;FOLD SLIN P253 Vel=2 m/s CPDAT253 Tool[4]:Microflown3D Base[2]:straight_sol;%{PE}
;FOLD Parameters ;%{h}
;Params IlfProvider=kukaroboter.basistech.inlineforms.movement.spline; Kuka.IsGlobalPoint=False; Kuka.PointName=P253; Kuka.BlendingEnabled=False; Kuka.MoveDataName=CPDAT253; Kuka.VelocityPath=2.000; Kuka.VelocityFieldEnabled=True; Kuka.ColDetectFieldEnabled=True; Kuka.CurrentCDSetIndex=0; Kuka.MovementParameterFieldEnabled=True; IlfCommand=SLIN
;ENDFOLD
SLIN XP253 WITH $VEL = SVEL_CP(2.0, , LCPDAT253),$TOOL = STOOL2(FP253),$BASE = SBASE(FP253.BASE_NO),$IPO_MODE = SIPO_MODE(FP253.IPO_FRAME),$LOAD = SLOAD(FP253.TOOL_NO),$ACC = SACC_CP(LCPDAT253),$ORI_TYPE = SORI_TYP(LCPDAT253),$APO = SAPO(LCPDAT253),$JERK = SJERK(LCPDAT253),$COLLMON_TOL_PRO[1] = USE_CM_PRO_VALUES(0)
;ENDFOLD

;FOLD SLIN P254 Vel=2 m/s CPDAT254 Tool[4]:Microflown3D Base[2]:straight_sol;%{PE}
;FOLD Parameters ;%{h}
;Params IlfProvider=kukaroboter.basistech.inlineforms.movement.spline; Kuka.IsGlobalPoint=False; Kuka.PointName=P254; Kuka.BlendingEnabled=False; Kuka.MoveDataName=CPDAT254; Kuka.VelocityPath=2.000; Kuka.VelocityFieldEnabled=True; Kuka.ColDetectFieldEnabled=True; Kuka.CurrentCDSetIndex=0; Kuka.MovementParameterFieldEnabled=True; IlfCommand=SLIN
;ENDFOLD
SLIN XP254 WITH $VEL = SVEL_CP(2.0, , LCPDAT254),$TOOL = STOOL2(FP254),$BASE = SBASE(FP254.BASE_NO),$IPO_MODE = SIPO_MODE(FP254.IPO_FRAME),$LOAD = SLOAD(FP254.TOOL_NO),$ACC = SACC_CP(LCPDAT254),$ORI_TYPE = SORI_TYP(LCPDAT254),$APO = SAPO(LCPDAT254),$JERK = SJERK(LCPDAT254),$COLLMON_TOL_PRO[1] = USE_CM_PRO_VALUES(0)
;ENDFOLD

;FOLD SLIN P255 Vel=2 m/s CPDAT255 Tool[4]:Microflown3D Base[2]:straight_sol;%{PE}
;FOLD Parameters ;%{h}
;Params IlfProvider=kukaroboter.basistech.inlineforms.movement.spline; Kuka.IsGlobalPoint=False; Kuka.PointName=P255; Kuka.BlendingEnabled=False; Kuka.MoveDataName=CPDAT255; Kuka.VelocityPath=2.000; Kuka.VelocityFieldEnabled=True; Kuka.ColDetectFieldEnabled=True; Kuka.CurrentCDSetIndex=0; Kuka.MovementParameterFieldEnabled=True; IlfCommand=SLIN
;ENDFOLD
SLIN XP255 WITH $VEL = SVEL_CP(2.0, , LCPDAT255),$TOOL = STOOL2(FP255),$BASE = SBASE(FP255.BASE_NO),$IPO_MODE = SIPO_MODE(FP255.IPO_FRAME),$LOAD = SLOAD(FP255.TOOL_NO),$ACC = SACC_CP(LCPDAT255),$ORI_TYPE = SORI_TYP(LCPDAT255),$APO = SAPO(LCPDAT255),$JERK = SJERK(LCPDAT255),$COLLMON_TOL_PRO[1] = USE_CM_PRO_VALUES(0)
;ENDFOLD

;FOLD SLIN P256 Vel=2 m/s CPDAT256 Tool[4]:Microflown3D Base[2]:straight_sol;%{PE}
;FOLD Parameters ;%{h}
;Params IlfProvider=kukaroboter.basistech.inlineforms.movement.spline; Kuka.IsGlobalPoint=False; Kuka.PointName=P256; Kuka.BlendingEnabled=False; Kuka.MoveDataName=CPDAT256; Kuka.VelocityPath=2.000; Kuka.VelocityFieldEnabled=True; Kuka.ColDetectFieldEnabled=True; Kuka.CurrentCDSetIndex=0; Kuka.MovementParameterFieldEnabled=True; IlfCommand=SLIN
;ENDFOLD
SLIN XP256 WITH $VEL = SVEL_CP(2.0, , LCPDAT256),$TOOL = STOOL2(FP256),$BASE = SBASE(FP256.BASE_NO),$IPO_MODE = SIPO_MODE(FP256.IPO_FRAME),$LOAD = SLOAD(FP256.TOOL_NO),$ACC = SACC_CP(LCPDAT256),$ORI_TYPE = SORI_TYP(LCPDAT256),$APO = SAPO(LCPDAT256),$JERK = SJERK(LCPDAT256),$COLLMON_TOL_PRO[1] = USE_CM_PRO_VALUES(0)
;ENDFOLD

;FOLD SLIN P257 Vel=2 m/s CPDAT257 Tool[4]:Microflown3D Base[2]:straight_sol;%{PE}
;FOLD Parameters ;%{h}
;Params IlfProvider=kukaroboter.basistech.inlineforms.movement.spline; Kuka.IsGlobalPoint=False; Kuka.PointName=P257; Kuka.BlendingEnabled=False; Kuka.MoveDataName=CPDAT257; Kuka.VelocityPath=2.000; Kuka.VelocityFieldEnabled=True; Kuka.ColDetectFieldEnabled=True; Kuka.CurrentCDSetIndex=0; Kuka.MovementParameterFieldEnabled=True; IlfCommand=SLIN
;ENDFOLD
SLIN XP257 WITH $VEL = SVEL_CP(2.0, , LCPDAT257),$TOOL = STOOL2(FP257),$BASE = SBASE(FP257.BASE_NO),$IPO_MODE = SIPO_MODE(FP257.IPO_FRAME),$LOAD = SLOAD(FP257.TOOL_NO),$ACC = SACC_CP(LCPDAT257),$ORI_TYPE = SORI_TYP(LCPDAT257),$APO = SAPO(LCPDAT257),$JERK = SJERK(LCPDAT257),$COLLMON_TOL_PRO[1] = USE_CM_PRO_VALUES(0)
;ENDFOLD

;FOLD SLIN P258 Vel=2 m/s CPDAT258 Tool[4]:Microflown3D Base[2]:straight_sol;%{PE}
;FOLD Parameters ;%{h}
;Params IlfProvider=kukaroboter.basistech.inlineforms.movement.spline; Kuka.IsGlobalPoint=False; Kuka.PointName=P258; Kuka.BlendingEnabled=False; Kuka.MoveDataName=CPDAT258; Kuka.VelocityPath=2.000; Kuka.VelocityFieldEnabled=True; Kuka.ColDetectFieldEnabled=True; Kuka.CurrentCDSetIndex=0; Kuka.MovementParameterFieldEnabled=True; IlfCommand=SLIN
;ENDFOLD
SLIN XP258 WITH $VEL = SVEL_CP(2.0, , LCPDAT258),$TOOL = STOOL2(FP258),$BASE = SBASE(FP258.BASE_NO),$IPO_MODE = SIPO_MODE(FP258.IPO_FRAME),$LOAD = SLOAD(FP258.TOOL_NO),$ACC = SACC_CP(LCPDAT258),$ORI_TYPE = SORI_TYP(LCPDAT258),$APO = SAPO(LCPDAT258),$JERK = SJERK(LCPDAT258),$COLLMON_TOL_PRO[1] = USE_CM_PRO_VALUES(0)
;ENDFOLD

;FOLD SLIN P259 Vel=2 m/s CPDAT259 Tool[4]:Microflown3D Base[2]:straight_sol;%{PE}
;FOLD Parameters ;%{h}
;Params IlfProvider=kukaroboter.basistech.inlineforms.movement.spline; Kuka.IsGlobalPoint=False; Kuka.PointName=P259; Kuka.BlendingEnabled=False; Kuka.MoveDataName=CPDAT259; Kuka.VelocityPath=2.000; Kuka.VelocityFieldEnabled=True; Kuka.ColDetectFieldEnabled=True; Kuka.CurrentCDSetIndex=0; Kuka.MovementParameterFieldEnabled=True; IlfCommand=SLIN
;ENDFOLD
SLIN XP259 WITH $VEL = SVEL_CP(2.0, , LCPDAT259),$TOOL = STOOL2(FP259),$BASE = SBASE(FP259.BASE_NO),$IPO_MODE = SIPO_MODE(FP259.IPO_FRAME),$LOAD = SLOAD(FP259.TOOL_NO),$ACC = SACC_CP(LCPDAT259),$ORI_TYPE = SORI_TYP(LCPDAT259),$APO = SAPO(LCPDAT259),$JERK = SJERK(LCPDAT259),$COLLMON_TOL_PRO[1] = USE_CM_PRO_VALUES(0)
;ENDFOLD

;FOLD SLIN P260 Vel=2 m/s CPDAT260 Tool[4]:Microflown3D Base[2]:straight_sol;%{PE}
;FOLD Parameters ;%{h}
;Params IlfProvider=kukaroboter.basistech.inlineforms.movement.spline; Kuka.IsGlobalPoint=False; Kuka.PointName=P260; Kuka.BlendingEnabled=False; Kuka.MoveDataName=CPDAT260; Kuka.VelocityPath=2.000; Kuka.VelocityFieldEnabled=True; Kuka.ColDetectFieldEnabled=True; Kuka.CurrentCDSetIndex=0; Kuka.MovementParameterFieldEnabled=True; IlfCommand=SLIN
;ENDFOLD
SLIN XP260 WITH $VEL = SVEL_CP(2.0, , LCPDAT260),$TOOL = STOOL2(FP260),$BASE = SBASE(FP260.BASE_NO),$IPO_MODE = SIPO_MODE(FP260.IPO_FRAME),$LOAD = SLOAD(FP260.TOOL_NO),$ACC = SACC_CP(LCPDAT260),$ORI_TYPE = SORI_TYP(LCPDAT260),$APO = SAPO(LCPDAT260),$JERK = SJERK(LCPDAT260),$COLLMON_TOL_PRO[1] = USE_CM_PRO_VALUES(0)
;ENDFOLD

;FOLD SLIN P261 Vel=2 m/s CPDAT261 Tool[4]:Microflown3D Base[2]:straight_sol;%{PE}
;FOLD Parameters ;%{h}
;Params IlfProvider=kukaroboter.basistech.inlineforms.movement.spline; Kuka.IsGlobalPoint=False; Kuka.PointName=P261; Kuka.BlendingEnabled=False; Kuka.MoveDataName=CPDAT261; Kuka.VelocityPath=2.000; Kuka.VelocityFieldEnabled=True; Kuka.ColDetectFieldEnabled=True; Kuka.CurrentCDSetIndex=0; Kuka.MovementParameterFieldEnabled=True; IlfCommand=SLIN
;ENDFOLD
SLIN XP261 WITH $VEL = SVEL_CP(2.0, , LCPDAT261),$TOOL = STOOL2(FP261),$BASE = SBASE(FP261.BASE_NO),$IPO_MODE = SIPO_MODE(FP261.IPO_FRAME),$LOAD = SLOAD(FP261.TOOL_NO),$ACC = SACC_CP(LCPDAT261),$ORI_TYPE = SORI_TYP(LCPDAT261),$APO = SAPO(LCPDAT261),$JERK = SJERK(LCPDAT261),$COLLMON_TOL_PRO[1] = USE_CM_PRO_VALUES(0)
;ENDFOLD

;FOLD SLIN P262 Vel=2 m/s CPDAT262 Tool[4]:Microflown3D Base[2]:straight_sol;%{PE}
;FOLD Parameters ;%{h}
;Params IlfProvider=kukaroboter.basistech.inlineforms.movement.spline; Kuka.IsGlobalPoint=False; Kuka.PointName=P262; Kuka.BlendingEnabled=False; Kuka.MoveDataName=CPDAT262; Kuka.VelocityPath=2.000; Kuka.VelocityFieldEnabled=True; Kuka.ColDetectFieldEnabled=True; Kuka.CurrentCDSetIndex=0; Kuka.MovementParameterFieldEnabled=True; IlfCommand=SLIN
;ENDFOLD
SLIN XP262 WITH $VEL = SVEL_CP(2.0, , LCPDAT262),$TOOL = STOOL2(FP262),$BASE = SBASE(FP262.BASE_NO),$IPO_MODE = SIPO_MODE(FP262.IPO_FRAME),$LOAD = SLOAD(FP262.TOOL_NO),$ACC = SACC_CP(LCPDAT262),$ORI_TYPE = SORI_TYP(LCPDAT262),$APO = SAPO(LCPDAT262),$JERK = SJERK(LCPDAT262),$COLLMON_TOL_PRO[1] = USE_CM_PRO_VALUES(0)
;ENDFOLD

;FOLD SLIN P263 Vel=2 m/s CPDAT263 Tool[4]:Microflown3D Base[2]:straight_sol;%{PE}
;FOLD Parameters ;%{h}
;Params IlfProvider=kukaroboter.basistech.inlineforms.movement.spline; Kuka.IsGlobalPoint=False; Kuka.PointName=P263; Kuka.BlendingEnabled=False; Kuka.MoveDataName=CPDAT263; Kuka.VelocityPath=2.000; Kuka.VelocityFieldEnabled=True; Kuka.ColDetectFieldEnabled=True; Kuka.CurrentCDSetIndex=0; Kuka.MovementParameterFieldEnabled=True; IlfCommand=SLIN
;ENDFOLD
SLIN XP263 WITH $VEL = SVEL_CP(2.0, , LCPDAT263),$TOOL = STOOL2(FP263),$BASE = SBASE(FP263.BASE_NO),$IPO_MODE = SIPO_MODE(FP263.IPO_FRAME),$LOAD = SLOAD(FP263.TOOL_NO),$ACC = SACC_CP(LCPDAT263),$ORI_TYPE = SORI_TYP(LCPDAT263),$APO = SAPO(LCPDAT263),$JERK = SJERK(LCPDAT263),$COLLMON_TOL_PRO[1] = USE_CM_PRO_VALUES(0)
;ENDFOLD

;FOLD SLIN P264 Vel=2 m/s CPDAT264 Tool[4]:Microflown3D Base[2]:straight_sol;%{PE}
;FOLD Parameters ;%{h}
;Params IlfProvider=kukaroboter.basistech.inlineforms.movement.spline; Kuka.IsGlobalPoint=False; Kuka.PointName=P264; Kuka.BlendingEnabled=False; Kuka.MoveDataName=CPDAT264; Kuka.VelocityPath=2.000; Kuka.VelocityFieldEnabled=True; Kuka.ColDetectFieldEnabled=True; Kuka.CurrentCDSetIndex=0; Kuka.MovementParameterFieldEnabled=True; IlfCommand=SLIN
;ENDFOLD
SLIN XP264 WITH $VEL = SVEL_CP(2.0, , LCPDAT264),$TOOL = STOOL2(FP264),$BASE = SBASE(FP264.BASE_NO),$IPO_MODE = SIPO_MODE(FP264.IPO_FRAME),$LOAD = SLOAD(FP264.TOOL_NO),$ACC = SACC_CP(LCPDAT264),$ORI_TYPE = SORI_TYP(LCPDAT264),$APO = SAPO(LCPDAT264),$JERK = SJERK(LCPDAT264),$COLLMON_TOL_PRO[1] = USE_CM_PRO_VALUES(0)
;ENDFOLD

;FOLD SLIN P265 Vel=2 m/s CPDAT265 Tool[4]:Microflown3D Base[2]:straight_sol;%{PE}
;FOLD Parameters ;%{h}
;Params IlfProvider=kukaroboter.basistech.inlineforms.movement.spline; Kuka.IsGlobalPoint=False; Kuka.PointName=P265; Kuka.BlendingEnabled=False; Kuka.MoveDataName=CPDAT265; Kuka.VelocityPath=2.000; Kuka.VelocityFieldEnabled=True; Kuka.ColDetectFieldEnabled=True; Kuka.CurrentCDSetIndex=0; Kuka.MovementParameterFieldEnabled=True; IlfCommand=SLIN
;ENDFOLD
SLIN XP265 WITH $VEL = SVEL_CP(2.0, , LCPDAT265),$TOOL = STOOL2(FP265),$BASE = SBASE(FP265.BASE_NO),$IPO_MODE = SIPO_MODE(FP265.IPO_FRAME),$LOAD = SLOAD(FP265.TOOL_NO),$ACC = SACC_CP(LCPDAT265),$ORI_TYPE = SORI_TYP(LCPDAT265),$APO = SAPO(LCPDAT265),$JERK = SJERK(LCPDAT265),$COLLMON_TOL_PRO[1] = USE_CM_PRO_VALUES(0)
;ENDFOLD

;FOLD SLIN P266 Vel=2 m/s CPDAT266 Tool[4]:Microflown3D Base[2]:straight_sol;%{PE}
;FOLD Parameters ;%{h}
;Params IlfProvider=kukaroboter.basistech.inlineforms.movement.spline; Kuka.IsGlobalPoint=False; Kuka.PointName=P266; Kuka.BlendingEnabled=False; Kuka.MoveDataName=CPDAT266; Kuka.VelocityPath=2.000; Kuka.VelocityFieldEnabled=True; Kuka.ColDetectFieldEnabled=True; Kuka.CurrentCDSetIndex=0; Kuka.MovementParameterFieldEnabled=True; IlfCommand=SLIN
;ENDFOLD
SLIN XP266 WITH $VEL = SVEL_CP(2.0, , LCPDAT266),$TOOL = STOOL2(FP266),$BASE = SBASE(FP266.BASE_NO),$IPO_MODE = SIPO_MODE(FP266.IPO_FRAME),$LOAD = SLOAD(FP266.TOOL_NO),$ACC = SACC_CP(LCPDAT266),$ORI_TYPE = SORI_TYP(LCPDAT266),$APO = SAPO(LCPDAT266),$JERK = SJERK(LCPDAT266),$COLLMON_TOL_PRO[1] = USE_CM_PRO_VALUES(0)
;ENDFOLD

;FOLD SLIN P267 Vel=2 m/s CPDAT267 Tool[4]:Microflown3D Base[2]:straight_sol;%{PE}
;FOLD Parameters ;%{h}
;Params IlfProvider=kukaroboter.basistech.inlineforms.movement.spline; Kuka.IsGlobalPoint=False; Kuka.PointName=P267; Kuka.BlendingEnabled=False; Kuka.MoveDataName=CPDAT267; Kuka.VelocityPath=2.000; Kuka.VelocityFieldEnabled=True; Kuka.ColDetectFieldEnabled=True; Kuka.CurrentCDSetIndex=0; Kuka.MovementParameterFieldEnabled=True; IlfCommand=SLIN
;ENDFOLD
SLIN XP267 WITH $VEL = SVEL_CP(2.0, , LCPDAT267),$TOOL = STOOL2(FP267),$BASE = SBASE(FP267.BASE_NO),$IPO_MODE = SIPO_MODE(FP267.IPO_FRAME),$LOAD = SLOAD(FP267.TOOL_NO),$ACC = SACC_CP(LCPDAT267),$ORI_TYPE = SORI_TYP(LCPDAT267),$APO = SAPO(LCPDAT267),$JERK = SJERK(LCPDAT267),$COLLMON_TOL_PRO[1] = USE_CM_PRO_VALUES(0)
;ENDFOLD

;FOLD SLIN P268 Vel=2 m/s CPDAT268 Tool[4]:Microflown3D Base[2]:straight_sol;%{PE}
;FOLD Parameters ;%{h}
;Params IlfProvider=kukaroboter.basistech.inlineforms.movement.spline; Kuka.IsGlobalPoint=False; Kuka.PointName=P268; Kuka.BlendingEnabled=False; Kuka.MoveDataName=CPDAT268; Kuka.VelocityPath=2.000; Kuka.VelocityFieldEnabled=True; Kuka.ColDetectFieldEnabled=True; Kuka.CurrentCDSetIndex=0; Kuka.MovementParameterFieldEnabled=True; IlfCommand=SLIN
;ENDFOLD
SLIN XP268 WITH $VEL = SVEL_CP(2.0, , LCPDAT268),$TOOL = STOOL2(FP268),$BASE = SBASE(FP268.BASE_NO),$IPO_MODE = SIPO_MODE(FP268.IPO_FRAME),$LOAD = SLOAD(FP268.TOOL_NO),$ACC = SACC_CP(LCPDAT268),$ORI_TYPE = SORI_TYP(LCPDAT268),$APO = SAPO(LCPDAT268),$JERK = SJERK(LCPDAT268),$COLLMON_TOL_PRO[1] = USE_CM_PRO_VALUES(0)
;ENDFOLD

;FOLD SLIN P269 Vel=2 m/s CPDAT269 Tool[4]:Microflown3D Base[2]:straight_sol;%{PE}
;FOLD Parameters ;%{h}
;Params IlfProvider=kukaroboter.basistech.inlineforms.movement.spline; Kuka.IsGlobalPoint=False; Kuka.PointName=P269; Kuka.BlendingEnabled=False; Kuka.MoveDataName=CPDAT269; Kuka.VelocityPath=2.000; Kuka.VelocityFieldEnabled=True; Kuka.ColDetectFieldEnabled=True; Kuka.CurrentCDSetIndex=0; Kuka.MovementParameterFieldEnabled=True; IlfCommand=SLIN
;ENDFOLD
SLIN XP269 WITH $VEL = SVEL_CP(2.0, , LCPDAT269),$TOOL = STOOL2(FP269),$BASE = SBASE(FP269.BASE_NO),$IPO_MODE = SIPO_MODE(FP269.IPO_FRAME),$LOAD = SLOAD(FP269.TOOL_NO),$ACC = SACC_CP(LCPDAT269),$ORI_TYPE = SORI_TYP(LCPDAT269),$APO = SAPO(LCPDAT269),$JERK = SJERK(LCPDAT269),$COLLMON_TOL_PRO[1] = USE_CM_PRO_VALUES(0)
;ENDFOLD

;FOLD SLIN P270 Vel=2 m/s CPDAT270 Tool[4]:Microflown3D Base[2]:straight_sol;%{PE}
;FOLD Parameters ;%{h}
;Params IlfProvider=kukaroboter.basistech.inlineforms.movement.spline; Kuka.IsGlobalPoint=False; Kuka.PointName=P270; Kuka.BlendingEnabled=False; Kuka.MoveDataName=CPDAT270; Kuka.VelocityPath=2.000; Kuka.VelocityFieldEnabled=True; Kuka.ColDetectFieldEnabled=True; Kuka.CurrentCDSetIndex=0; Kuka.MovementParameterFieldEnabled=True; IlfCommand=SLIN
;ENDFOLD
SLIN XP270 WITH $VEL = SVEL_CP(2.0, , LCPDAT270),$TOOL = STOOL2(FP270),$BASE = SBASE(FP270.BASE_NO),$IPO_MODE = SIPO_MODE(FP270.IPO_FRAME),$LOAD = SLOAD(FP270.TOOL_NO),$ACC = SACC_CP(LCPDAT270),$ORI_TYPE = SORI_TYP(LCPDAT270),$APO = SAPO(LCPDAT270),$JERK = SJERK(LCPDAT270),$COLLMON_TOL_PRO[1] = USE_CM_PRO_VALUES(0)
;ENDFOLD

;FOLD SLIN P271 Vel=1 m/s CPDAT271 Tool[4]:Microflown3D Base[2]:straight_sol;%{PE}
;FOLD Parameters ;%{h}
;Params IlfProvider=kukaroboter.basistech.inlineforms.movement.spline; Kuka.IsGlobalPoint=False; Kuka.PointName=P271; Kuka.BlendingEnabled=False; Kuka.MoveDataName=CPDAT271; Kuka.VelocityPath=1.000; Kuka.VelocityFieldEnabled=True; Kuka.ColDetectFieldEnabled=True; Kuka.CurrentCDSetIndex=0; Kuka.MovementParameterFieldEnabled=True; IlfCommand=SLIN
;ENDFOLD
SLIN XP271 WITH $VEL = SVEL_CP(2.0, , LCPDAT271),$TOOL = STOOL2(FP271),$BASE = SBASE(FP271.BASE_NO),$IPO_MODE = SIPO_MODE(FP271.IPO_FRAME),$LOAD = SLOAD(FP271.TOOL_NO),$ACC = SACC_CP(LCPDAT271),$ORI_TYPE = SORI_TYP(LCPDAT271),$APO = SAPO(LCPDAT271),$JERK = SJERK(LCPDAT271),$COLLMON_TOL_PRO[1] = USE_CM_PRO_VALUES(0)
;ENDFOLD

;FOLD SLIN P272 Vel=1 m/s CPDAT272 Tool[4]:Microflown3D Base[2]:straight_sol;%{PE}
;FOLD Parameters ;%{h}
;Params IlfProvider=kukaroboter.basistech.inlineforms.movement.spline; Kuka.IsGlobalPoint=False; Kuka.PointName=P272; Kuka.BlendingEnabled=False; Kuka.MoveDataName=CPDAT272; Kuka.VelocityPath=1.000; Kuka.VelocityFieldEnabled=True; Kuka.ColDetectFieldEnabled=True; Kuka.CurrentCDSetIndex=0; Kuka.MovementParameterFieldEnabled=True; IlfCommand=SLIN
;ENDFOLD
SLIN XP272 WITH $VEL = SVEL_CP(2.0, , LCPDAT272),$TOOL = STOOL2(FP272),$BASE = SBASE(FP272.BASE_NO),$IPO_MODE = SIPO_MODE(FP272.IPO_FRAME),$LOAD = SLOAD(FP272.TOOL_NO),$ACC = SACC_CP(LCPDAT272),$ORI_TYPE = SORI_TYP(LCPDAT272),$APO = SAPO(LCPDAT272),$JERK = SJERK(LCPDAT272),$COLLMON_TOL_PRO[1] = USE_CM_PRO_VALUES(0)
;ENDFOLD

;FOLD SLIN P273 Vel=2 m/s CPDAT273 Tool[4]:Microflown3D Base[2]:straight_sol;%{PE}
;FOLD Parameters ;%{h}
;Params IlfProvider=kukaroboter.basistech.inlineforms.movement.spline; Kuka.IsGlobalPoint=False; Kuka.PointName=P273; Kuka.BlendingEnabled=False; Kuka.MoveDataName=CPDAT273; Kuka.VelocityPath=2.000; Kuka.VelocityFieldEnabled=True; Kuka.ColDetectFieldEnabled=True; Kuka.CurrentCDSetIndex=0; Kuka.MovementParameterFieldEnabled=True; IlfCommand=SLIN
;ENDFOLD
SLIN XP273 WITH $VEL = SVEL_CP(2.0, , LCPDAT273),$TOOL = STOOL2(FP273),$BASE = SBASE(FP273.BASE_NO),$IPO_MODE = SIPO_MODE(FP273.IPO_FRAME),$LOAD = SLOAD(FP273.TOOL_NO),$ACC = SACC_CP(LCPDAT273),$ORI_TYPE = SORI_TYP(LCPDAT273),$APO = SAPO(LCPDAT273),$JERK = SJERK(LCPDAT273),$COLLMON_TOL_PRO[1] = USE_CM_PRO_VALUES(0)
;ENDFOLD

;FOLD SLIN P274 Vel=2 m/s CPDAT274 Tool[4]:Microflown3D Base[2]:straight_sol;%{PE}
;FOLD Parameters ;%{h}
;Params IlfProvider=kukaroboter.basistech.inlineforms.movement.spline; Kuka.IsGlobalPoint=False; Kuka.PointName=P274; Kuka.BlendingEnabled=False; Kuka.MoveDataName=CPDAT274; Kuka.VelocityPath=2.000; Kuka.VelocityFieldEnabled=True; Kuka.ColDetectFieldEnabled=True; Kuka.CurrentCDSetIndex=0; Kuka.MovementParameterFieldEnabled=True; IlfCommand=SLIN
;ENDFOLD
SLIN XP274 WITH $VEL = SVEL_CP(2.0, , LCPDAT274),$TOOL = STOOL2(FP274),$BASE = SBASE(FP274.BASE_NO),$IPO_MODE = SIPO_MODE(FP274.IPO_FRAME),$LOAD = SLOAD(FP274.TOOL_NO),$ACC = SACC_CP(LCPDAT274),$ORI_TYPE = SORI_TYP(LCPDAT274),$APO = SAPO(LCPDAT274),$JERK = SJERK(LCPDAT274),$COLLMON_TOL_PRO[1] = USE_CM_PRO_VALUES(0)
;ENDFOLD

;FOLD SLIN P275 Vel=2 m/s CPDAT275 Tool[4]:Microflown3D Base[2]:straight_sol;%{PE}
;FOLD Parameters ;%{h}
;Params IlfProvider=kukaroboter.basistech.inlineforms.movement.spline; Kuka.IsGlobalPoint=False; Kuka.PointName=P275; Kuka.BlendingEnabled=False; Kuka.MoveDataName=CPDAT275; Kuka.VelocityPath=2.000; Kuka.VelocityFieldEnabled=True; Kuka.ColDetectFieldEnabled=True; Kuka.CurrentCDSetIndex=0; Kuka.MovementParameterFieldEnabled=True; IlfCommand=SLIN
;ENDFOLD
SLIN XP275 WITH $VEL = SVEL_CP(2.0, , LCPDAT275),$TOOL = STOOL2(FP275),$BASE = SBASE(FP275.BASE_NO),$IPO_MODE = SIPO_MODE(FP275.IPO_FRAME),$LOAD = SLOAD(FP275.TOOL_NO),$ACC = SACC_CP(LCPDAT275),$ORI_TYPE = SORI_TYP(LCPDAT275),$APO = SAPO(LCPDAT275),$JERK = SJERK(LCPDAT275),$COLLMON_TOL_PRO[1] = USE_CM_PRO_VALUES(0)
;ENDFOLD

;FOLD SLIN P276 Vel=2 m/s CPDAT276 Tool[4]:Microflown3D Base[2]:straight_sol;%{PE}
;FOLD Parameters ;%{h}
;Params IlfProvider=kukaroboter.basistech.inlineforms.movement.spline; Kuka.IsGlobalPoint=False; Kuka.PointName=P276; Kuka.BlendingEnabled=False; Kuka.MoveDataName=CPDAT276; Kuka.VelocityPath=2.000; Kuka.VelocityFieldEnabled=True; Kuka.ColDetectFieldEnabled=True; Kuka.CurrentCDSetIndex=0; Kuka.MovementParameterFieldEnabled=True; IlfCommand=SLIN
;ENDFOLD
SLIN XP276 WITH $VEL = SVEL_CP(2.0, , LCPDAT276),$TOOL = STOOL2(FP276),$BASE = SBASE(FP276.BASE_NO),$IPO_MODE = SIPO_MODE(FP276.IPO_FRAME),$LOAD = SLOAD(FP276.TOOL_NO),$ACC = SACC_CP(LCPDAT276),$ORI_TYPE = SORI_TYP(LCPDAT276),$APO = SAPO(LCPDAT276),$JERK = SJERK(LCPDAT276),$COLLMON_TOL_PRO[1] = USE_CM_PRO_VALUES(0)
;ENDFOLD

;FOLD SLIN P277 Vel=2 m/s CPDAT277 Tool[4]:Microflown3D Base[2]:straight_sol;%{PE}
;FOLD Parameters ;%{h}
;Params IlfProvider=kukaroboter.basistech.inlineforms.movement.spline; Kuka.IsGlobalPoint=False; Kuka.PointName=P277; Kuka.BlendingEnabled=False; Kuka.MoveDataName=CPDAT277; Kuka.VelocityPath=2.000; Kuka.VelocityFieldEnabled=True; Kuka.ColDetectFieldEnabled=True; Kuka.CurrentCDSetIndex=0; Kuka.MovementParameterFieldEnabled=True; IlfCommand=SLIN
;ENDFOLD
SLIN XP277 WITH $VEL = SVEL_CP(2.0, , LCPDAT277),$TOOL = STOOL2(FP277),$BASE = SBASE(FP277.BASE_NO),$IPO_MODE = SIPO_MODE(FP277.IPO_FRAME),$LOAD = SLOAD(FP277.TOOL_NO),$ACC = SACC_CP(LCPDAT277),$ORI_TYPE = SORI_TYP(LCPDAT277),$APO = SAPO(LCPDAT277),$JERK = SJERK(LCPDAT277),$COLLMON_TOL_PRO[1] = USE_CM_PRO_VALUES(0)
;ENDFOLD

;FOLD SLIN P278 Vel=2 m/s CPDAT278 Tool[4]:Microflown3D Base[2]:straight_sol;%{PE}
;FOLD Parameters ;%{h}
;Params IlfProvider=kukaroboter.basistech.inlineforms.movement.spline; Kuka.IsGlobalPoint=False; Kuka.PointName=P278; Kuka.BlendingEnabled=False; Kuka.MoveDataName=CPDAT278; Kuka.VelocityPath=2.000; Kuka.VelocityFieldEnabled=True; Kuka.ColDetectFieldEnabled=True; Kuka.CurrentCDSetIndex=0; Kuka.MovementParameterFieldEnabled=True; IlfCommand=SLIN
;ENDFOLD
SLIN XP278 WITH $VEL = SVEL_CP(2.0, , LCPDAT278),$TOOL = STOOL2(FP278),$BASE = SBASE(FP278.BASE_NO),$IPO_MODE = SIPO_MODE(FP278.IPO_FRAME),$LOAD = SLOAD(FP278.TOOL_NO),$ACC = SACC_CP(LCPDAT278),$ORI_TYPE = SORI_TYP(LCPDAT278),$APO = SAPO(LCPDAT278),$JERK = SJERK(LCPDAT278),$COLLMON_TOL_PRO[1] = USE_CM_PRO_VALUES(0)
;ENDFOLD

;FOLD SLIN P279 Vel=2 m/s CPDAT279 Tool[4]:Microflown3D Base[2]:straight_sol;%{PE}
;FOLD Parameters ;%{h}
;Params IlfProvider=kukaroboter.basistech.inlineforms.movement.spline; Kuka.IsGlobalPoint=False; Kuka.PointName=P279; Kuka.BlendingEnabled=False; Kuka.MoveDataName=CPDAT279; Kuka.VelocityPath=2.000; Kuka.VelocityFieldEnabled=True; Kuka.ColDetectFieldEnabled=True; Kuka.CurrentCDSetIndex=0; Kuka.MovementParameterFieldEnabled=True; IlfCommand=SLIN
;ENDFOLD
SLIN XP279 WITH $VEL = SVEL_CP(2.0, , LCPDAT279),$TOOL = STOOL2(FP279),$BASE = SBASE(FP279.BASE_NO),$IPO_MODE = SIPO_MODE(FP279.IPO_FRAME),$LOAD = SLOAD(FP279.TOOL_NO),$ACC = SACC_CP(LCPDAT279),$ORI_TYPE = SORI_TYP(LCPDAT279),$APO = SAPO(LCPDAT279),$JERK = SJERK(LCPDAT279),$COLLMON_TOL_PRO[1] = USE_CM_PRO_VALUES(0)
;ENDFOLD

;FOLD SLIN P280 Vel=2 m/s CPDAT280 Tool[4]:Microflown3D Base[2]:straight_sol;%{PE}
;FOLD Parameters ;%{h}
;Params IlfProvider=kukaroboter.basistech.inlineforms.movement.spline; Kuka.IsGlobalPoint=False; Kuka.PointName=P280; Kuka.BlendingEnabled=False; Kuka.MoveDataName=CPDAT280; Kuka.VelocityPath=2.000; Kuka.VelocityFieldEnabled=True; Kuka.ColDetectFieldEnabled=True; Kuka.CurrentCDSetIndex=0; Kuka.MovementParameterFieldEnabled=True; IlfCommand=SLIN
;ENDFOLD
SLIN XP280 WITH $VEL = SVEL_CP(2.0, , LCPDAT280),$TOOL = STOOL2(FP280),$BASE = SBASE(FP280.BASE_NO),$IPO_MODE = SIPO_MODE(FP280.IPO_FRAME),$LOAD = SLOAD(FP280.TOOL_NO),$ACC = SACC_CP(LCPDAT280),$ORI_TYPE = SORI_TYP(LCPDAT280),$APO = SAPO(LCPDAT280),$JERK = SJERK(LCPDAT280),$COLLMON_TOL_PRO[1] = USE_CM_PRO_VALUES(0)
;ENDFOLD

;FOLD SLIN P281 Vel=2 m/s CPDAT281 Tool[4]:Microflown3D Base[2]:straight_sol;%{PE}
;FOLD Parameters ;%{h}
;Params IlfProvider=kukaroboter.basistech.inlineforms.movement.spline; Kuka.IsGlobalPoint=False; Kuka.PointName=P281; Kuka.BlendingEnabled=False; Kuka.MoveDataName=CPDAT281; Kuka.VelocityPath=2.000; Kuka.VelocityFieldEnabled=True; Kuka.ColDetectFieldEnabled=True; Kuka.CurrentCDSetIndex=0; Kuka.MovementParameterFieldEnabled=True; IlfCommand=SLIN
;ENDFOLD
SLIN XP281 WITH $VEL = SVEL_CP(2.0, , LCPDAT281),$TOOL = STOOL2(FP281),$BASE = SBASE(FP281.BASE_NO),$IPO_MODE = SIPO_MODE(FP281.IPO_FRAME),$LOAD = SLOAD(FP281.TOOL_NO),$ACC = SACC_CP(LCPDAT281),$ORI_TYPE = SORI_TYP(LCPDAT281),$APO = SAPO(LCPDAT281),$JERK = SJERK(LCPDAT281),$COLLMON_TOL_PRO[1] = USE_CM_PRO_VALUES(0)
;ENDFOLD

;FOLD SLIN P282 Vel=2 m/s CPDAT282 Tool[4]:Microflown3D Base[2]:straight_sol;%{PE}
;FOLD Parameters ;%{h}
;Params IlfProvider=kukaroboter.basistech.inlineforms.movement.spline; Kuka.IsGlobalPoint=False; Kuka.PointName=P282; Kuka.BlendingEnabled=False; Kuka.MoveDataName=CPDAT282; Kuka.VelocityPath=2.000; Kuka.VelocityFieldEnabled=True; Kuka.ColDetectFieldEnabled=True; Kuka.CurrentCDSetIndex=0; Kuka.MovementParameterFieldEnabled=True; IlfCommand=SLIN
;ENDFOLD
SLIN XP282 WITH $VEL = SVEL_CP(2.0, , LCPDAT282),$TOOL = STOOL2(FP282),$BASE = SBASE(FP282.BASE_NO),$IPO_MODE = SIPO_MODE(FP282.IPO_FRAME),$LOAD = SLOAD(FP282.TOOL_NO),$ACC = SACC_CP(LCPDAT282),$ORI_TYPE = SORI_TYP(LCPDAT282),$APO = SAPO(LCPDAT282),$JERK = SJERK(LCPDAT282),$COLLMON_TOL_PRO[1] = USE_CM_PRO_VALUES(0)
;ENDFOLD

;FOLD SLIN P283 Vel=2 m/s CPDAT283 Tool[4]:Microflown3D Base[2]:straight_sol;%{PE}
;FOLD Parameters ;%{h}
;Params IlfProvider=kukaroboter.basistech.inlineforms.movement.spline; Kuka.IsGlobalPoint=False; Kuka.PointName=P283; Kuka.BlendingEnabled=False; Kuka.MoveDataName=CPDAT283; Kuka.VelocityPath=2.000; Kuka.VelocityFieldEnabled=True; Kuka.ColDetectFieldEnabled=True; Kuka.CurrentCDSetIndex=0; Kuka.MovementParameterFieldEnabled=True; IlfCommand=SLIN
;ENDFOLD
SLIN XP283 WITH $VEL = SVEL_CP(2.0, , LCPDAT283),$TOOL = STOOL2(FP283),$BASE = SBASE(FP283.BASE_NO),$IPO_MODE = SIPO_MODE(FP283.IPO_FRAME),$LOAD = SLOAD(FP283.TOOL_NO),$ACC = SACC_CP(LCPDAT283),$ORI_TYPE = SORI_TYP(LCPDAT283),$APO = SAPO(LCPDAT283),$JERK = SJERK(LCPDAT283),$COLLMON_TOL_PRO[1] = USE_CM_PRO_VALUES(0)
;ENDFOLD

;FOLD SLIN P284 Vel=2 m/s CPDAT284 Tool[4]:Microflown3D Base[2]:straight_sol;%{PE}
;FOLD Parameters ;%{h}
;Params IlfProvider=kukaroboter.basistech.inlineforms.movement.spline; Kuka.IsGlobalPoint=False; Kuka.PointName=P284; Kuka.BlendingEnabled=False; Kuka.MoveDataName=CPDAT284; Kuka.VelocityPath=2.000; Kuka.VelocityFieldEnabled=True; Kuka.ColDetectFieldEnabled=True; Kuka.CurrentCDSetIndex=0; Kuka.MovementParameterFieldEnabled=True; IlfCommand=SLIN
;ENDFOLD
SLIN XP284 WITH $VEL = SVEL_CP(2.0, , LCPDAT284),$TOOL = STOOL2(FP284),$BASE = SBASE(FP284.BASE_NO),$IPO_MODE = SIPO_MODE(FP284.IPO_FRAME),$LOAD = SLOAD(FP284.TOOL_NO),$ACC = SACC_CP(LCPDAT284),$ORI_TYPE = SORI_TYP(LCPDAT284),$APO = SAPO(LCPDAT284),$JERK = SJERK(LCPDAT284),$COLLMON_TOL_PRO[1] = USE_CM_PRO_VALUES(0)
;ENDFOLD

;FOLD SLIN P285 Vel=2 m/s CPDAT285 Tool[4]:Microflown3D Base[2]:straight_sol;%{PE}
;FOLD Parameters ;%{h}
;Params IlfProvider=kukaroboter.basistech.inlineforms.movement.spline; Kuka.IsGlobalPoint=False; Kuka.PointName=P285; Kuka.BlendingEnabled=False; Kuka.MoveDataName=CPDAT285; Kuka.VelocityPath=2.000; Kuka.VelocityFieldEnabled=True; Kuka.ColDetectFieldEnabled=True; Kuka.CurrentCDSetIndex=0; Kuka.MovementParameterFieldEnabled=True; IlfCommand=SLIN
;ENDFOLD
SLIN XP285 WITH $VEL = SVEL_CP(2.0, , LCPDAT285),$TOOL = STOOL2(FP285),$BASE = SBASE(FP285.BASE_NO),$IPO_MODE = SIPO_MODE(FP285.IPO_FRAME),$LOAD = SLOAD(FP285.TOOL_NO),$ACC = SACC_CP(LCPDAT285),$ORI_TYPE = SORI_TYP(LCPDAT285),$APO = SAPO(LCPDAT285),$JERK = SJERK(LCPDAT285),$COLLMON_TOL_PRO[1] = USE_CM_PRO_VALUES(0)
;ENDFOLD

;FOLD SLIN P286 Vel=2 m/s CPDAT286 Tool[4]:Microflown3D Base[2]:straight_sol;%{PE}
;FOLD Parameters ;%{h}
;Params IlfProvider=kukaroboter.basistech.inlineforms.movement.spline; Kuka.IsGlobalPoint=False; Kuka.PointName=P286; Kuka.BlendingEnabled=False; Kuka.MoveDataName=CPDAT286; Kuka.VelocityPath=2.000; Kuka.VelocityFieldEnabled=True; Kuka.ColDetectFieldEnabled=True; Kuka.CurrentCDSetIndex=0; Kuka.MovementParameterFieldEnabled=True; IlfCommand=SLIN
;ENDFOLD
SLIN XP286 WITH $VEL = SVEL_CP(2.0, , LCPDAT286),$TOOL = STOOL2(FP286),$BASE = SBASE(FP286.BASE_NO),$IPO_MODE = SIPO_MODE(FP286.IPO_FRAME),$LOAD = SLOAD(FP286.TOOL_NO),$ACC = SACC_CP(LCPDAT286),$ORI_TYPE = SORI_TYP(LCPDAT286),$APO = SAPO(LCPDAT286),$JERK = SJERK(LCPDAT286),$COLLMON_TOL_PRO[1] = USE_CM_PRO_VALUES(0)
;ENDFOLD

;FOLD SLIN P287 Vel=2 m/s CPDAT287 Tool[4]:Microflown3D Base[2]:straight_sol;%{PE}
;FOLD Parameters ;%{h}
;Params IlfProvider=kukaroboter.basistech.inlineforms.movement.spline; Kuka.IsGlobalPoint=False; Kuka.PointName=P287; Kuka.BlendingEnabled=False; Kuka.MoveDataName=CPDAT287; Kuka.VelocityPath=2.000; Kuka.VelocityFieldEnabled=True; Kuka.ColDetectFieldEnabled=True; Kuka.CurrentCDSetIndex=0; Kuka.MovementParameterFieldEnabled=True; IlfCommand=SLIN
;ENDFOLD
SLIN XP287 WITH $VEL = SVEL_CP(2.0, , LCPDAT287),$TOOL = STOOL2(FP287),$BASE = SBASE(FP287.BASE_NO),$IPO_MODE = SIPO_MODE(FP287.IPO_FRAME),$LOAD = SLOAD(FP287.TOOL_NO),$ACC = SACC_CP(LCPDAT287),$ORI_TYPE = SORI_TYP(LCPDAT287),$APO = SAPO(LCPDAT287),$JERK = SJERK(LCPDAT287),$COLLMON_TOL_PRO[1] = USE_CM_PRO_VALUES(0)
;ENDFOLD

;FOLD SLIN P288 Vel=2 m/s CPDAT288 Tool[4]:Microflown3D Base[2]:straight_sol;%{PE}
;FOLD Parameters ;%{h}
;Params IlfProvider=kukaroboter.basistech.inlineforms.movement.spline; Kuka.IsGlobalPoint=False; Kuka.PointName=P288; Kuka.BlendingEnabled=False; Kuka.MoveDataName=CPDAT288; Kuka.VelocityPath=2.000; Kuka.VelocityFieldEnabled=True; Kuka.ColDetectFieldEnabled=True; Kuka.CurrentCDSetIndex=0; Kuka.MovementParameterFieldEnabled=True; IlfCommand=SLIN
;ENDFOLD
SLIN XP288 WITH $VEL = SVEL_CP(2.0, , LCPDAT288),$TOOL = STOOL2(FP288),$BASE = SBASE(FP288.BASE_NO),$IPO_MODE = SIPO_MODE(FP288.IPO_FRAME),$LOAD = SLOAD(FP288.TOOL_NO),$ACC = SACC_CP(LCPDAT288),$ORI_TYPE = SORI_TYP(LCPDAT288),$APO = SAPO(LCPDAT288),$JERK = SJERK(LCPDAT288),$COLLMON_TOL_PRO[1] = USE_CM_PRO_VALUES(0)
;ENDFOLD

;FOLD SLIN P289 Vel=2 m/s CPDAT289 Tool[4]:Microflown3D Base[2]:straight_sol;%{PE}
;FOLD Parameters ;%{h}
;Params IlfProvider=kukaroboter.basistech.inlineforms.movement.spline; Kuka.IsGlobalPoint=False; Kuka.PointName=P289; Kuka.BlendingEnabled=False; Kuka.MoveDataName=CPDAT289; Kuka.VelocityPath=2.000; Kuka.VelocityFieldEnabled=True; Kuka.ColDetectFieldEnabled=True; Kuka.CurrentCDSetIndex=0; Kuka.MovementParameterFieldEnabled=True; IlfCommand=SLIN
;ENDFOLD
SLIN XP289 WITH $VEL = SVEL_CP(2.0, , LCPDAT289),$TOOL = STOOL2(FP289),$BASE = SBASE(FP289.BASE_NO),$IPO_MODE = SIPO_MODE(FP289.IPO_FRAME),$LOAD = SLOAD(FP289.TOOL_NO),$ACC = SACC_CP(LCPDAT289),$ORI_TYPE = SORI_TYP(LCPDAT289),$APO = SAPO(LCPDAT289),$JERK = SJERK(LCPDAT289),$COLLMON_TOL_PRO[1] = USE_CM_PRO_VALUES(0)
;ENDFOLD

;FOLD SLIN P290 Vel=2 m/s CPDAT290 Tool[4]:Microflown3D Base[2]:straight_sol;%{PE}
;FOLD Parameters ;%{h}
;Params IlfProvider=kukaroboter.basistech.inlineforms.movement.spline; Kuka.IsGlobalPoint=False; Kuka.PointName=P290; Kuka.BlendingEnabled=False; Kuka.MoveDataName=CPDAT290; Kuka.VelocityPath=2.000; Kuka.VelocityFieldEnabled=True; Kuka.ColDetectFieldEnabled=True; Kuka.CurrentCDSetIndex=0; Kuka.MovementParameterFieldEnabled=True; IlfCommand=SLIN
;ENDFOLD
SLIN XP290 WITH $VEL = SVEL_CP(2.0, , LCPDAT290),$TOOL = STOOL2(FP290),$BASE = SBASE(FP290.BASE_NO),$IPO_MODE = SIPO_MODE(FP290.IPO_FRAME),$LOAD = SLOAD(FP290.TOOL_NO),$ACC = SACC_CP(LCPDAT290),$ORI_TYPE = SORI_TYP(LCPDAT290),$APO = SAPO(LCPDAT290),$JERK = SJERK(LCPDAT290),$COLLMON_TOL_PRO[1] = USE_CM_PRO_VALUES(0)
;ENDFOLD

;FOLD SLIN P291 Vel=2 m/s CPDAT291 Tool[4]:Microflown3D Base[2]:straight_sol;%{PE}
;FOLD Parameters ;%{h}
;Params IlfProvider=kukaroboter.basistech.inlineforms.movement.spline; Kuka.IsGlobalPoint=False; Kuka.PointName=P291; Kuka.BlendingEnabled=False; Kuka.MoveDataName=CPDAT291; Kuka.VelocityPath=2.000; Kuka.VelocityFieldEnabled=True; Kuka.ColDetectFieldEnabled=True; Kuka.CurrentCDSetIndex=0; Kuka.MovementParameterFieldEnabled=True; IlfCommand=SLIN
;ENDFOLD
SLIN XP291 WITH $VEL = SVEL_CP(2.0, , LCPDAT291),$TOOL = STOOL2(FP291),$BASE = SBASE(FP291.BASE_NO),$IPO_MODE = SIPO_MODE(FP291.IPO_FRAME),$LOAD = SLOAD(FP291.TOOL_NO),$ACC = SACC_CP(LCPDAT291),$ORI_TYPE = SORI_TYP(LCPDAT291),$APO = SAPO(LCPDAT291),$JERK = SJERK(LCPDAT291),$COLLMON_TOL_PRO[1] = USE_CM_PRO_VALUES(0)
;ENDFOLD

;FOLD SLIN P292 Vel=2 m/s CPDAT292 Tool[4]:Microflown3D Base[2]:straight_sol;%{PE}
;FOLD Parameters ;%{h}
;Params IlfProvider=kukaroboter.basistech.inlineforms.movement.spline; Kuka.IsGlobalPoint=False; Kuka.PointName=P292; Kuka.BlendingEnabled=False; Kuka.MoveDataName=CPDAT292; Kuka.VelocityPath=2.000; Kuka.VelocityFieldEnabled=True; Kuka.ColDetectFieldEnabled=True; Kuka.CurrentCDSetIndex=0; Kuka.MovementParameterFieldEnabled=True; IlfCommand=SLIN
;ENDFOLD
SLIN XP292 WITH $VEL = SVEL_CP(2.0, , LCPDAT292),$TOOL = STOOL2(FP292),$BASE = SBASE(FP292.BASE_NO),$IPO_MODE = SIPO_MODE(FP292.IPO_FRAME),$LOAD = SLOAD(FP292.TOOL_NO),$ACC = SACC_CP(LCPDAT292),$ORI_TYPE = SORI_TYP(LCPDAT292),$APO = SAPO(LCPDAT292),$JERK = SJERK(LCPDAT292),$COLLMON_TOL_PRO[1] = USE_CM_PRO_VALUES(0)
;ENDFOLD

;FOLD SLIN P293 Vel=2 m/s CPDAT293 Tool[4]:Microflown3D Base[2]:straight_sol;%{PE}
;FOLD Parameters ;%{h}
;Params IlfProvider=kukaroboter.basistech.inlineforms.movement.spline; Kuka.IsGlobalPoint=False; Kuka.PointName=P293; Kuka.BlendingEnabled=False; Kuka.MoveDataName=CPDAT293; Kuka.VelocityPath=2.000; Kuka.VelocityFieldEnabled=True; Kuka.ColDetectFieldEnabled=True; Kuka.CurrentCDSetIndex=0; Kuka.MovementParameterFieldEnabled=True; IlfCommand=SLIN
;ENDFOLD
SLIN XP293 WITH $VEL = SVEL_CP(2.0, , LCPDAT293),$TOOL = STOOL2(FP293),$BASE = SBASE(FP293.BASE_NO),$IPO_MODE = SIPO_MODE(FP293.IPO_FRAME),$LOAD = SLOAD(FP293.TOOL_NO),$ACC = SACC_CP(LCPDAT293),$ORI_TYPE = SORI_TYP(LCPDAT293),$APO = SAPO(LCPDAT293),$JERK = SJERK(LCPDAT293),$COLLMON_TOL_PRO[1] = USE_CM_PRO_VALUES(0)
;ENDFOLD

;FOLD SLIN P294 Vel=2 m/s CPDAT294 Tool[4]:Microflown3D Base[2]:straight_sol;%{PE}
;FOLD Parameters ;%{h}
;Params IlfProvider=kukaroboter.basistech.inlineforms.movement.spline; Kuka.IsGlobalPoint=False; Kuka.PointName=P294; Kuka.BlendingEnabled=False; Kuka.MoveDataName=CPDAT294; Kuka.VelocityPath=2.000; Kuka.VelocityFieldEnabled=True; Kuka.ColDetectFieldEnabled=True; Kuka.CurrentCDSetIndex=0; Kuka.MovementParameterFieldEnabled=True; IlfCommand=SLIN
;ENDFOLD
SLIN XP294 WITH $VEL = SVEL_CP(2.0, , LCPDAT294),$TOOL = STOOL2(FP294),$BASE = SBASE(FP294.BASE_NO),$IPO_MODE = SIPO_MODE(FP294.IPO_FRAME),$LOAD = SLOAD(FP294.TOOL_NO),$ACC = SACC_CP(LCPDAT294),$ORI_TYPE = SORI_TYP(LCPDAT294),$APO = SAPO(LCPDAT294),$JERK = SJERK(LCPDAT294),$COLLMON_TOL_PRO[1] = USE_CM_PRO_VALUES(0)
;ENDFOLD

;FOLD SLIN P295 Vel=2 m/s CPDAT295 Tool[4]:Microflown3D Base[2]:straight_sol;%{PE}
;FOLD Parameters ;%{h}
;Params IlfProvider=kukaroboter.basistech.inlineforms.movement.spline; Kuka.IsGlobalPoint=False; Kuka.PointName=P295; Kuka.BlendingEnabled=False; Kuka.MoveDataName=CPDAT295; Kuka.VelocityPath=2.000; Kuka.VelocityFieldEnabled=True; Kuka.ColDetectFieldEnabled=True; Kuka.CurrentCDSetIndex=0; Kuka.MovementParameterFieldEnabled=True; IlfCommand=SLIN
;ENDFOLD
SLIN XP295 WITH $VEL = SVEL_CP(2.0, , LCPDAT295),$TOOL = STOOL2(FP295),$BASE = SBASE(FP295.BASE_NO),$IPO_MODE = SIPO_MODE(FP295.IPO_FRAME),$LOAD = SLOAD(FP295.TOOL_NO),$ACC = SACC_CP(LCPDAT295),$ORI_TYPE = SORI_TYP(LCPDAT295),$APO = SAPO(LCPDAT295),$JERK = SJERK(LCPDAT295),$COLLMON_TOL_PRO[1] = USE_CM_PRO_VALUES(0)
;ENDFOLD

;FOLD SLIN P296 Vel=2 m/s CPDAT296 Tool[4]:Microflown3D Base[2]:straight_sol;%{PE}
;FOLD Parameters ;%{h}
;Params IlfProvider=kukaroboter.basistech.inlineforms.movement.spline; Kuka.IsGlobalPoint=False; Kuka.PointName=P296; Kuka.BlendingEnabled=False; Kuka.MoveDataName=CPDAT296; Kuka.VelocityPath=2.000; Kuka.VelocityFieldEnabled=True; Kuka.ColDetectFieldEnabled=True; Kuka.CurrentCDSetIndex=0; Kuka.MovementParameterFieldEnabled=True; IlfCommand=SLIN
;ENDFOLD
SLIN XP296 WITH $VEL = SVEL_CP(2.0, , LCPDAT296),$TOOL = STOOL2(FP296),$BASE = SBASE(FP296.BASE_NO),$IPO_MODE = SIPO_MODE(FP296.IPO_FRAME),$LOAD = SLOAD(FP296.TOOL_NO),$ACC = SACC_CP(LCPDAT296),$ORI_TYPE = SORI_TYP(LCPDAT296),$APO = SAPO(LCPDAT296),$JERK = SJERK(LCPDAT296),$COLLMON_TOL_PRO[1] = USE_CM_PRO_VALUES(0)
;ENDFOLD

;FOLD SLIN P297 Vel=2 m/s CPDAT297 Tool[4]:Microflown3D Base[2]:straight_sol;%{PE}
;FOLD Parameters ;%{h}
;Params IlfProvider=kukaroboter.basistech.inlineforms.movement.spline; Kuka.IsGlobalPoint=False; Kuka.PointName=P297; Kuka.BlendingEnabled=False; Kuka.MoveDataName=CPDAT297; Kuka.VelocityPath=2.000; Kuka.VelocityFieldEnabled=True; Kuka.ColDetectFieldEnabled=True; Kuka.CurrentCDSetIndex=0; Kuka.MovementParameterFieldEnabled=True; IlfCommand=SLIN
;ENDFOLD
SLIN XP297 WITH $VEL = SVEL_CP(2.0, , LCPDAT297),$TOOL = STOOL2(FP297),$BASE = SBASE(FP297.BASE_NO),$IPO_MODE = SIPO_MODE(FP297.IPO_FRAME),$LOAD = SLOAD(FP297.TOOL_NO),$ACC = SACC_CP(LCPDAT297),$ORI_TYPE = SORI_TYP(LCPDAT297),$APO = SAPO(LCPDAT297),$JERK = SJERK(LCPDAT297),$COLLMON_TOL_PRO[1] = USE_CM_PRO_VALUES(0)
;ENDFOLD

;FOLD SLIN P298 Vel=2 m/s CPDAT298 Tool[4]:Microflown3D Base[2]:straight_sol;%{PE}
;FOLD Parameters ;%{h}
;Params IlfProvider=kukaroboter.basistech.inlineforms.movement.spline; Kuka.IsGlobalPoint=False; Kuka.PointName=P298; Kuka.BlendingEnabled=False; Kuka.MoveDataName=CPDAT298; Kuka.VelocityPath=2.000; Kuka.VelocityFieldEnabled=True; Kuka.ColDetectFieldEnabled=True; Kuka.CurrentCDSetIndex=0; Kuka.MovementParameterFieldEnabled=True; IlfCommand=SLIN
;ENDFOLD
SLIN XP298 WITH $VEL = SVEL_CP(2.0, , LCPDAT298),$TOOL = STOOL2(FP298),$BASE = SBASE(FP298.BASE_NO),$IPO_MODE = SIPO_MODE(FP298.IPO_FRAME),$LOAD = SLOAD(FP298.TOOL_NO),$ACC = SACC_CP(LCPDAT298),$ORI_TYPE = SORI_TYP(LCPDAT298),$APO = SAPO(LCPDAT298),$JERK = SJERK(LCPDAT298),$COLLMON_TOL_PRO[1] = USE_CM_PRO_VALUES(0)
;ENDFOLD

;FOLD SLIN P299 Vel=2 m/s CPDAT299 Tool[4]:Microflown3D Base[2]:straight_sol;%{PE}
;FOLD Parameters ;%{h}
;Params IlfProvider=kukaroboter.basistech.inlineforms.movement.spline; Kuka.IsGlobalPoint=False; Kuka.PointName=P299; Kuka.BlendingEnabled=False; Kuka.MoveDataName=CPDAT299; Kuka.VelocityPath=2.000; Kuka.VelocityFieldEnabled=True; Kuka.ColDetectFieldEnabled=True; Kuka.CurrentCDSetIndex=0; Kuka.MovementParameterFieldEnabled=True; IlfCommand=SLIN
;ENDFOLD
SLIN XP299 WITH $VEL = SVEL_CP(2.0, , LCPDAT299),$TOOL = STOOL2(FP299),$BASE = SBASE(FP299.BASE_NO),$IPO_MODE = SIPO_MODE(FP299.IPO_FRAME),$LOAD = SLOAD(FP299.TOOL_NO),$ACC = SACC_CP(LCPDAT299),$ORI_TYPE = SORI_TYP(LCPDAT299),$APO = SAPO(LCPDAT299),$JERK = SJERK(LCPDAT299),$COLLMON_TOL_PRO[1] = USE_CM_PRO_VALUES(0)
;ENDFOLD

;FOLD SLIN P300 Vel=2 m/s CPDAT300 Tool[4]:Microflown3D Base[2]:straight_sol;%{PE}
;FOLD Parameters ;%{h}
;Params IlfProvider=kukaroboter.basistech.inlineforms.movement.spline; Kuka.IsGlobalPoint=False; Kuka.PointName=P300; Kuka.BlendingEnabled=False; Kuka.MoveDataName=CPDAT300; Kuka.VelocityPath=2.000; Kuka.VelocityFieldEnabled=True; Kuka.ColDetectFieldEnabled=True; Kuka.CurrentCDSetIndex=0; Kuka.MovementParameterFieldEnabled=True; IlfCommand=SLIN
;ENDFOLD
SLIN XP300 WITH $VEL = SVEL_CP(2.0, , LCPDAT300),$TOOL = STOOL2(FP300),$BASE = SBASE(FP300.BASE_NO),$IPO_MODE = SIPO_MODE(FP300.IPO_FRAME),$LOAD = SLOAD(FP300.TOOL_NO),$ACC = SACC_CP(LCPDAT300),$ORI_TYPE = SORI_TYP(LCPDAT300),$APO = SAPO(LCPDAT300),$JERK = SJERK(LCPDAT300),$COLLMON_TOL_PRO[1] = USE_CM_PRO_VALUES(0)
;ENDFOLD

;FOLD SLIN P301 Vel=2 m/s CPDAT301 Tool[4]:Microflown3D Base[2]:straight_sol;%{PE}
;FOLD Parameters ;%{h}
;Params IlfProvider=kukaroboter.basistech.inlineforms.movement.spline; Kuka.IsGlobalPoint=False; Kuka.PointName=P301; Kuka.BlendingEnabled=False; Kuka.MoveDataName=CPDAT301; Kuka.VelocityPath=2.000; Kuka.VelocityFieldEnabled=True; Kuka.ColDetectFieldEnabled=True; Kuka.CurrentCDSetIndex=0; Kuka.MovementParameterFieldEnabled=True; IlfCommand=SLIN
;ENDFOLD
SLIN XP301 WITH $VEL = SVEL_CP(2.0, , LCPDAT301),$TOOL = STOOL2(FP301),$BASE = SBASE(FP301.BASE_NO),$IPO_MODE = SIPO_MODE(FP301.IPO_FRAME),$LOAD = SLOAD(FP301.TOOL_NO),$ACC = SACC_CP(LCPDAT301),$ORI_TYPE = SORI_TYP(LCPDAT301),$APO = SAPO(LCPDAT301),$JERK = SJERK(LCPDAT301),$COLLMON_TOL_PRO[1] = USE_CM_PRO_VALUES(0)
;ENDFOLD

;FOLD SLIN P302 Vel=2 m/s CPDAT302 Tool[4]:Microflown3D Base[2]:straight_sol;%{PE}
;FOLD Parameters ;%{h}
;Params IlfProvider=kukaroboter.basistech.inlineforms.movement.spline; Kuka.IsGlobalPoint=False; Kuka.PointName=P302; Kuka.BlendingEnabled=False; Kuka.MoveDataName=CPDAT302; Kuka.VelocityPath=2.000; Kuka.VelocityFieldEnabled=True; Kuka.ColDetectFieldEnabled=True; Kuka.CurrentCDSetIndex=0; Kuka.MovementParameterFieldEnabled=True; IlfCommand=SLIN
;ENDFOLD
SLIN XP302 WITH $VEL = SVEL_CP(2.0, , LCPDAT302),$TOOL = STOOL2(FP302),$BASE = SBASE(FP302.BASE_NO),$IPO_MODE = SIPO_MODE(FP302.IPO_FRAME),$LOAD = SLOAD(FP302.TOOL_NO),$ACC = SACC_CP(LCPDAT302),$ORI_TYPE = SORI_TYP(LCPDAT302),$APO = SAPO(LCPDAT302),$JERK = SJERK(LCPDAT302),$COLLMON_TOL_PRO[1] = USE_CM_PRO_VALUES(0)
;ENDFOLD

;FOLD SLIN P303 Vel=2 m/s CPDAT303 Tool[4]:Microflown3D Base[2]:straight_sol;%{PE}
;FOLD Parameters ;%{h}
;Params IlfProvider=kukaroboter.basistech.inlineforms.movement.spline; Kuka.IsGlobalPoint=False; Kuka.PointName=P303; Kuka.BlendingEnabled=False; Kuka.MoveDataName=CPDAT303; Kuka.VelocityPath=2.000; Kuka.VelocityFieldEnabled=True; Kuka.ColDetectFieldEnabled=True; Kuka.CurrentCDSetIndex=0; Kuka.MovementParameterFieldEnabled=True; IlfCommand=SLIN
;ENDFOLD
SLIN XP303 WITH $VEL = SVEL_CP(2.0, , LCPDAT303),$TOOL = STOOL2(FP303),$BASE = SBASE(FP303.BASE_NO),$IPO_MODE = SIPO_MODE(FP303.IPO_FRAME),$LOAD = SLOAD(FP303.TOOL_NO),$ACC = SACC_CP(LCPDAT303),$ORI_TYPE = SORI_TYP(LCPDAT303),$APO = SAPO(LCPDAT303),$JERK = SJERK(LCPDAT303),$COLLMON_TOL_PRO[1] = USE_CM_PRO_VALUES(0)
;ENDFOLD

;FOLD SLIN P304 Vel=2 m/s CPDAT304 Tool[4]:Microflown3D Base[2]:straight_sol;%{PE}
;FOLD Parameters ;%{h}
;Params IlfProvider=kukaroboter.basistech.inlineforms.movement.spline; Kuka.IsGlobalPoint=False; Kuka.PointName=P304; Kuka.BlendingEnabled=False; Kuka.MoveDataName=CPDAT304; Kuka.VelocityPath=2.000; Kuka.VelocityFieldEnabled=True; Kuka.ColDetectFieldEnabled=True; Kuka.CurrentCDSetIndex=0; Kuka.MovementParameterFieldEnabled=True; IlfCommand=SLIN
;ENDFOLD
SLIN XP304 WITH $VEL = SVEL_CP(2.0, , LCPDAT304),$TOOL = STOOL2(FP304),$BASE = SBASE(FP304.BASE_NO),$IPO_MODE = SIPO_MODE(FP304.IPO_FRAME),$LOAD = SLOAD(FP304.TOOL_NO),$ACC = SACC_CP(LCPDAT304),$ORI_TYPE = SORI_TYP(LCPDAT304),$APO = SAPO(LCPDAT304),$JERK = SJERK(LCPDAT304),$COLLMON_TOL_PRO[1] = USE_CM_PRO_VALUES(0)
;ENDFOLD

;FOLD SLIN P305 Vel=2 m/s CPDAT305 Tool[4]:Microflown3D Base[2]:straight_sol;%{PE}
;FOLD Parameters ;%{h}
;Params IlfProvider=kukaroboter.basistech.inlineforms.movement.spline; Kuka.IsGlobalPoint=False; Kuka.PointName=P305; Kuka.BlendingEnabled=False; Kuka.MoveDataName=CPDAT305; Kuka.VelocityPath=2.000; Kuka.VelocityFieldEnabled=True; Kuka.ColDetectFieldEnabled=True; Kuka.CurrentCDSetIndex=0; Kuka.MovementParameterFieldEnabled=True; IlfCommand=SLIN
;ENDFOLD
SLIN XP305 WITH $VEL = SVEL_CP(2.0, , LCPDAT305),$TOOL = STOOL2(FP305),$BASE = SBASE(FP305.BASE_NO),$IPO_MODE = SIPO_MODE(FP305.IPO_FRAME),$LOAD = SLOAD(FP305.TOOL_NO),$ACC = SACC_CP(LCPDAT305),$ORI_TYPE = SORI_TYP(LCPDAT305),$APO = SAPO(LCPDAT305),$JERK = SJERK(LCPDAT305),$COLLMON_TOL_PRO[1] = USE_CM_PRO_VALUES(0)
;ENDFOLD

;FOLD SLIN P306 Vel=2 m/s CPDAT306 Tool[4]:Microflown3D Base[2]:straight_sol;%{PE}
;FOLD Parameters ;%{h}
;Params IlfProvider=kukaroboter.basistech.inlineforms.movement.spline; Kuka.IsGlobalPoint=False; Kuka.PointName=P306; Kuka.BlendingEnabled=False; Kuka.MoveDataName=CPDAT306; Kuka.VelocityPath=2.000; Kuka.VelocityFieldEnabled=True; Kuka.ColDetectFieldEnabled=True; Kuka.CurrentCDSetIndex=0; Kuka.MovementParameterFieldEnabled=True; IlfCommand=SLIN
;ENDFOLD
SLIN XP306 WITH $VEL = SVEL_CP(2.0, , LCPDAT306),$TOOL = STOOL2(FP306),$BASE = SBASE(FP306.BASE_NO),$IPO_MODE = SIPO_MODE(FP306.IPO_FRAME),$LOAD = SLOAD(FP306.TOOL_NO),$ACC = SACC_CP(LCPDAT306),$ORI_TYPE = SORI_TYP(LCPDAT306),$APO = SAPO(LCPDAT306),$JERK = SJERK(LCPDAT306),$COLLMON_TOL_PRO[1] = USE_CM_PRO_VALUES(0)
;ENDFOLD

;FOLD SLIN P307 Vel=2 m/s CPDAT307 Tool[4]:Microflown3D Base[2]:straight_sol;%{PE}
;FOLD Parameters ;%{h}
;Params IlfProvider=kukaroboter.basistech.inlineforms.movement.spline; Kuka.IsGlobalPoint=False; Kuka.PointName=P307; Kuka.BlendingEnabled=False; Kuka.MoveDataName=CPDAT307; Kuka.VelocityPath=2.000; Kuka.VelocityFieldEnabled=True; Kuka.ColDetectFieldEnabled=True; Kuka.CurrentCDSetIndex=0; Kuka.MovementParameterFieldEnabled=True; IlfCommand=SLIN
;ENDFOLD
SLIN XP307 WITH $VEL = SVEL_CP(2.0, , LCPDAT307),$TOOL = STOOL2(FP307),$BASE = SBASE(FP307.BASE_NO),$IPO_MODE = SIPO_MODE(FP307.IPO_FRAME),$LOAD = SLOAD(FP307.TOOL_NO),$ACC = SACC_CP(LCPDAT307),$ORI_TYPE = SORI_TYP(LCPDAT307),$APO = SAPO(LCPDAT307),$JERK = SJERK(LCPDAT307),$COLLMON_TOL_PRO[1] = USE_CM_PRO_VALUES(0)
;ENDFOLD

;FOLD SLIN P308 Vel=2 m/s CPDAT308 Tool[4]:Microflown3D Base[2]:straight_sol;%{PE}
;FOLD Parameters ;%{h}
;Params IlfProvider=kukaroboter.basistech.inlineforms.movement.spline; Kuka.IsGlobalPoint=False; Kuka.PointName=P308; Kuka.BlendingEnabled=False; Kuka.MoveDataName=CPDAT308; Kuka.VelocityPath=2.000; Kuka.VelocityFieldEnabled=True; Kuka.ColDetectFieldEnabled=True; Kuka.CurrentCDSetIndex=0; Kuka.MovementParameterFieldEnabled=True; IlfCommand=SLIN
;ENDFOLD
SLIN XP308 WITH $VEL = SVEL_CP(2.0, , LCPDAT308),$TOOL = STOOL2(FP308),$BASE = SBASE(FP308.BASE_NO),$IPO_MODE = SIPO_MODE(FP308.IPO_FRAME),$LOAD = SLOAD(FP308.TOOL_NO),$ACC = SACC_CP(LCPDAT308),$ORI_TYPE = SORI_TYP(LCPDAT308),$APO = SAPO(LCPDAT308),$JERK = SJERK(LCPDAT308),$COLLMON_TOL_PRO[1] = USE_CM_PRO_VALUES(0)
;ENDFOLD

;FOLD SLIN P309 Vel=2 m/s CPDAT309 Tool[4]:Microflown3D Base[2]:straight_sol;%{PE}
;FOLD Parameters ;%{h}
;Params IlfProvider=kukaroboter.basistech.inlineforms.movement.spline; Kuka.IsGlobalPoint=False; Kuka.PointName=P309; Kuka.BlendingEnabled=False; Kuka.MoveDataName=CPDAT309; Kuka.VelocityPath=2.000; Kuka.VelocityFieldEnabled=True; Kuka.ColDetectFieldEnabled=True; Kuka.CurrentCDSetIndex=0; Kuka.MovementParameterFieldEnabled=True; IlfCommand=SLIN
;ENDFOLD
SLIN XP309 WITH $VEL = SVEL_CP(2.0, , LCPDAT309),$TOOL = STOOL2(FP309),$BASE = SBASE(FP309.BASE_NO),$IPO_MODE = SIPO_MODE(FP309.IPO_FRAME),$LOAD = SLOAD(FP309.TOOL_NO),$ACC = SACC_CP(LCPDAT309),$ORI_TYPE = SORI_TYP(LCPDAT309),$APO = SAPO(LCPDAT309),$JERK = SJERK(LCPDAT309),$COLLMON_TOL_PRO[1] = USE_CM_PRO_VALUES(0)
;ENDFOLD

;FOLD SLIN P310 Vel=2 m/s CPDAT310 Tool[4]:Microflown3D Base[2]:straight_sol;%{PE}
;FOLD Parameters ;%{h}
;Params IlfProvider=kukaroboter.basistech.inlineforms.movement.spline; Kuka.IsGlobalPoint=False; Kuka.PointName=P310; Kuka.BlendingEnabled=False; Kuka.MoveDataName=CPDAT310; Kuka.VelocityPath=2.000; Kuka.VelocityFieldEnabled=True; Kuka.ColDetectFieldEnabled=True; Kuka.CurrentCDSetIndex=0; Kuka.MovementParameterFieldEnabled=True; IlfCommand=SLIN
;ENDFOLD
SLIN XP310 WITH $VEL = SVEL_CP(2.0, , LCPDAT310),$TOOL = STOOL2(FP310),$BASE = SBASE(FP310.BASE_NO),$IPO_MODE = SIPO_MODE(FP310.IPO_FRAME),$LOAD = SLOAD(FP310.TOOL_NO),$ACC = SACC_CP(LCPDAT310),$ORI_TYPE = SORI_TYP(LCPDAT310),$APO = SAPO(LCPDAT310),$JERK = SJERK(LCPDAT310),$COLLMON_TOL_PRO[1] = USE_CM_PRO_VALUES(0)
;ENDFOLD

;FOLD SLIN P311 Vel=2 m/s CPDAT311 Tool[4]:Microflown3D Base[2]:straight_sol;%{PE}
;FOLD Parameters ;%{h}
;Params IlfProvider=kukaroboter.basistech.inlineforms.movement.spline; Kuka.IsGlobalPoint=False; Kuka.PointName=P311; Kuka.BlendingEnabled=False; Kuka.MoveDataName=CPDAT311; Kuka.VelocityPath=2.000; Kuka.VelocityFieldEnabled=True; Kuka.ColDetectFieldEnabled=True; Kuka.CurrentCDSetIndex=0; Kuka.MovementParameterFieldEnabled=True; IlfCommand=SLIN
;ENDFOLD
SLIN XP311 WITH $VEL = SVEL_CP(2.0, , LCPDAT311),$TOOL = STOOL2(FP311),$BASE = SBASE(FP311.BASE_NO),$IPO_MODE = SIPO_MODE(FP311.IPO_FRAME),$LOAD = SLOAD(FP311.TOOL_NO),$ACC = SACC_CP(LCPDAT311),$ORI_TYPE = SORI_TYP(LCPDAT311),$APO = SAPO(LCPDAT311),$JERK = SJERK(LCPDAT311),$COLLMON_TOL_PRO[1] = USE_CM_PRO_VALUES(0)
;ENDFOLD

;FOLD SLIN P312 Vel=2 m/s CPDAT312 Tool[4]:Microflown3D Base[2]:straight_sol;%{PE}
;FOLD Parameters ;%{h}
;Params IlfProvider=kukaroboter.basistech.inlineforms.movement.spline; Kuka.IsGlobalPoint=False; Kuka.PointName=P312; Kuka.BlendingEnabled=False; Kuka.MoveDataName=CPDAT312; Kuka.VelocityPath=2.000; Kuka.VelocityFieldEnabled=True; Kuka.ColDetectFieldEnabled=True; Kuka.CurrentCDSetIndex=0; Kuka.MovementParameterFieldEnabled=True; IlfCommand=SLIN
;ENDFOLD
SLIN XP312 WITH $VEL = SVEL_CP(2.0, , LCPDAT312),$TOOL = STOOL2(FP312),$BASE = SBASE(FP312.BASE_NO),$IPO_MODE = SIPO_MODE(FP312.IPO_FRAME),$LOAD = SLOAD(FP312.TOOL_NO),$ACC = SACC_CP(LCPDAT312),$ORI_TYPE = SORI_TYP(LCPDAT312),$APO = SAPO(LCPDAT312),$JERK = SJERK(LCPDAT312),$COLLMON_TOL_PRO[1] = USE_CM_PRO_VALUES(0)
;ENDFOLD

;FOLD SLIN P313 Vel=2 m/s CPDAT313 Tool[4]:Microflown3D Base[2]:straight_sol;%{PE}
;FOLD Parameters ;%{h}
;Params IlfProvider=kukaroboter.basistech.inlineforms.movement.spline; Kuka.IsGlobalPoint=False; Kuka.PointName=P313; Kuka.BlendingEnabled=False; Kuka.MoveDataName=CPDAT313; Kuka.VelocityPath=2.000; Kuka.VelocityFieldEnabled=True; Kuka.ColDetectFieldEnabled=True; Kuka.CurrentCDSetIndex=0; Kuka.MovementParameterFieldEnabled=True; IlfCommand=SLIN
;ENDFOLD
SLIN XP313 WITH $VEL = SVEL_CP(2.0, , LCPDAT313),$TOOL = STOOL2(FP313),$BASE = SBASE(FP313.BASE_NO),$IPO_MODE = SIPO_MODE(FP313.IPO_FRAME),$LOAD = SLOAD(FP313.TOOL_NO),$ACC = SACC_CP(LCPDAT313),$ORI_TYPE = SORI_TYP(LCPDAT313),$APO = SAPO(LCPDAT313),$JERK = SJERK(LCPDAT313),$COLLMON_TOL_PRO[1] = USE_CM_PRO_VALUES(0)
;ENDFOLD

;FOLD SLIN P314 Vel=2 m/s CPDAT314 Tool[4]:Microflown3D Base[2]:straight_sol;%{PE}
;FOLD Parameters ;%{h}
;Params IlfProvider=kukaroboter.basistech.inlineforms.movement.spline; Kuka.IsGlobalPoint=False; Kuka.PointName=P314; Kuka.BlendingEnabled=False; Kuka.MoveDataName=CPDAT314; Kuka.VelocityPath=2.000; Kuka.VelocityFieldEnabled=True; Kuka.ColDetectFieldEnabled=True; Kuka.CurrentCDSetIndex=0; Kuka.MovementParameterFieldEnabled=True; IlfCommand=SLIN
;ENDFOLD
SLIN XP314 WITH $VEL = SVEL_CP(2.0, , LCPDAT314),$TOOL = STOOL2(FP314),$BASE = SBASE(FP314.BASE_NO),$IPO_MODE = SIPO_MODE(FP314.IPO_FRAME),$LOAD = SLOAD(FP314.TOOL_NO),$ACC = SACC_CP(LCPDAT314),$ORI_TYPE = SORI_TYP(LCPDAT314),$APO = SAPO(LCPDAT314),$JERK = SJERK(LCPDAT314),$COLLMON_TOL_PRO[1] = USE_CM_PRO_VALUES(0)
;ENDFOLD

;FOLD SLIN P315 Vel=2 m/s CPDAT315 Tool[4]:Microflown3D Base[2]:straight_sol;%{PE}
;FOLD Parameters ;%{h}
;Params IlfProvider=kukaroboter.basistech.inlineforms.movement.spline; Kuka.IsGlobalPoint=False; Kuka.PointName=P315; Kuka.BlendingEnabled=False; Kuka.MoveDataName=CPDAT315; Kuka.VelocityPath=2.000; Kuka.VelocityFieldEnabled=True; Kuka.ColDetectFieldEnabled=True; Kuka.CurrentCDSetIndex=0; Kuka.MovementParameterFieldEnabled=True; IlfCommand=SLIN
;ENDFOLD
SLIN XP315 WITH $VEL = SVEL_CP(2.0, , LCPDAT315),$TOOL = STOOL2(FP315),$BASE = SBASE(FP315.BASE_NO),$IPO_MODE = SIPO_MODE(FP315.IPO_FRAME),$LOAD = SLOAD(FP315.TOOL_NO),$ACC = SACC_CP(LCPDAT315),$ORI_TYPE = SORI_TYP(LCPDAT315),$APO = SAPO(LCPDAT315),$JERK = SJERK(LCPDAT315),$COLLMON_TOL_PRO[1] = USE_CM_PRO_VALUES(0)
;ENDFOLD

;FOLD SLIN P316 Vel=2 m/s CPDAT316 Tool[4]:Microflown3D Base[2]:straight_sol;%{PE}
;FOLD Parameters ;%{h}
;Params IlfProvider=kukaroboter.basistech.inlineforms.movement.spline; Kuka.IsGlobalPoint=False; Kuka.PointName=P316; Kuka.BlendingEnabled=False; Kuka.MoveDataName=CPDAT316; Kuka.VelocityPath=2.000; Kuka.VelocityFieldEnabled=True; Kuka.ColDetectFieldEnabled=True; Kuka.CurrentCDSetIndex=0; Kuka.MovementParameterFieldEnabled=True; IlfCommand=SLIN
;ENDFOLD
SLIN XP316 WITH $VEL = SVEL_CP(2.0, , LCPDAT316),$TOOL = STOOL2(FP316),$BASE = SBASE(FP316.BASE_NO),$IPO_MODE = SIPO_MODE(FP316.IPO_FRAME),$LOAD = SLOAD(FP316.TOOL_NO),$ACC = SACC_CP(LCPDAT316),$ORI_TYPE = SORI_TYP(LCPDAT316),$APO = SAPO(LCPDAT316),$JERK = SJERK(LCPDAT316),$COLLMON_TOL_PRO[1] = USE_CM_PRO_VALUES(0)
;ENDFOLD

;FOLD SLIN P317 Vel=2 m/s CPDAT317 Tool[4]:Microflown3D Base[2]:straight_sol;%{PE}
;FOLD Parameters ;%{h}
;Params IlfProvider=kukaroboter.basistech.inlineforms.movement.spline; Kuka.IsGlobalPoint=False; Kuka.PointName=P317; Kuka.BlendingEnabled=False; Kuka.MoveDataName=CPDAT317; Kuka.VelocityPath=2.000; Kuka.VelocityFieldEnabled=True; Kuka.ColDetectFieldEnabled=True; Kuka.CurrentCDSetIndex=0; Kuka.MovementParameterFieldEnabled=True; IlfCommand=SLIN
;ENDFOLD
SLIN XP317 WITH $VEL = SVEL_CP(2.0, , LCPDAT317),$TOOL = STOOL2(FP317),$BASE = SBASE(FP317.BASE_NO),$IPO_MODE = SIPO_MODE(FP317.IPO_FRAME),$LOAD = SLOAD(FP317.TOOL_NO),$ACC = SACC_CP(LCPDAT317),$ORI_TYPE = SORI_TYP(LCPDAT317),$APO = SAPO(LCPDAT317),$JERK = SJERK(LCPDAT317),$COLLMON_TOL_PRO[1] = USE_CM_PRO_VALUES(0)
;ENDFOLD

;FOLD SLIN P318 Vel=2 m/s CPDAT318 Tool[4]:Microflown3D Base[2]:straight_sol;%{PE}
;FOLD Parameters ;%{h}
;Params IlfProvider=kukaroboter.basistech.inlineforms.movement.spline; Kuka.IsGlobalPoint=False; Kuka.PointName=P318; Kuka.BlendingEnabled=False; Kuka.MoveDataName=CPDAT318; Kuka.VelocityPath=2.000; Kuka.VelocityFieldEnabled=True; Kuka.ColDetectFieldEnabled=True; Kuka.CurrentCDSetIndex=0; Kuka.MovementParameterFieldEnabled=True; IlfCommand=SLIN
;ENDFOLD
SLIN XP318 WITH $VEL = SVEL_CP(2.0, , LCPDAT318),$TOOL = STOOL2(FP318),$BASE = SBASE(FP318.BASE_NO),$IPO_MODE = SIPO_MODE(FP318.IPO_FRAME),$LOAD = SLOAD(FP318.TOOL_NO),$ACC = SACC_CP(LCPDAT318),$ORI_TYPE = SORI_TYP(LCPDAT318),$APO = SAPO(LCPDAT318),$JERK = SJERK(LCPDAT318),$COLLMON_TOL_PRO[1] = USE_CM_PRO_VALUES(0)
;ENDFOLD

;FOLD SLIN P319 Vel=2 m/s CPDAT319 Tool[4]:Microflown3D Base[2]:straight_sol;%{PE}
;FOLD Parameters ;%{h}
;Params IlfProvider=kukaroboter.basistech.inlineforms.movement.spline; Kuka.IsGlobalPoint=False; Kuka.PointName=P319; Kuka.BlendingEnabled=False; Kuka.MoveDataName=CPDAT319; Kuka.VelocityPath=2.000; Kuka.VelocityFieldEnabled=True; Kuka.ColDetectFieldEnabled=True; Kuka.CurrentCDSetIndex=0; Kuka.MovementParameterFieldEnabled=True; IlfCommand=SLIN
;ENDFOLD
SLIN XP319 WITH $VEL = SVEL_CP(2.0, , LCPDAT319),$TOOL = STOOL2(FP319),$BASE = SBASE(FP319.BASE_NO),$IPO_MODE = SIPO_MODE(FP319.IPO_FRAME),$LOAD = SLOAD(FP319.TOOL_NO),$ACC = SACC_CP(LCPDAT319),$ORI_TYPE = SORI_TYP(LCPDAT319),$APO = SAPO(LCPDAT319),$JERK = SJERK(LCPDAT319),$COLLMON_TOL_PRO[1] = USE_CM_PRO_VALUES(0)
;ENDFOLD

;FOLD SLIN P320 Vel=2 m/s CPDAT320 Tool[4]:Microflown3D Base[2]:straight_sol;%{PE}
;FOLD Parameters ;%{h}
;Params IlfProvider=kukaroboter.basistech.inlineforms.movement.spline; Kuka.IsGlobalPoint=False; Kuka.PointName=P320; Kuka.BlendingEnabled=False; Kuka.MoveDataName=CPDAT320; Kuka.VelocityPath=2.000; Kuka.VelocityFieldEnabled=True; Kuka.ColDetectFieldEnabled=True; Kuka.CurrentCDSetIndex=0; Kuka.MovementParameterFieldEnabled=True; IlfCommand=SLIN
;ENDFOLD
SLIN XP320 WITH $VEL = SVEL_CP(2.0, , LCPDAT320),$TOOL = STOOL2(FP320),$BASE = SBASE(FP320.BASE_NO),$IPO_MODE = SIPO_MODE(FP320.IPO_FRAME),$LOAD = SLOAD(FP320.TOOL_NO),$ACC = SACC_CP(LCPDAT320),$ORI_TYPE = SORI_TYP(LCPDAT320),$APO = SAPO(LCPDAT320),$JERK = SJERK(LCPDAT320),$COLLMON_TOL_PRO[1] = USE_CM_PRO_VALUES(0)
;ENDFOLD

;FOLD SLIN P321 Vel=2 m/s CPDAT321 Tool[4]:Microflown3D Base[2]:straight_sol;%{PE}
;FOLD Parameters ;%{h}
;Params IlfProvider=kukaroboter.basistech.inlineforms.movement.spline; Kuka.IsGlobalPoint=False; Kuka.PointName=P321; Kuka.BlendingEnabled=False; Kuka.MoveDataName=CPDAT321; Kuka.VelocityPath=2.000; Kuka.VelocityFieldEnabled=True; Kuka.ColDetectFieldEnabled=True; Kuka.CurrentCDSetIndex=0; Kuka.MovementParameterFieldEnabled=True; IlfCommand=SLIN
;ENDFOLD
SLIN XP321 WITH $VEL = SVEL_CP(2.0, , LCPDAT321),$TOOL = STOOL2(FP321),$BASE = SBASE(FP321.BASE_NO),$IPO_MODE = SIPO_MODE(FP321.IPO_FRAME),$LOAD = SLOAD(FP321.TOOL_NO),$ACC = SACC_CP(LCPDAT321),$ORI_TYPE = SORI_TYP(LCPDAT321),$APO = SAPO(LCPDAT321),$JERK = SJERK(LCPDAT321),$COLLMON_TOL_PRO[1] = USE_CM_PRO_VALUES(0)
;ENDFOLD

;FOLD SLIN P322 Vel=2 m/s CPDAT322 Tool[4]:Microflown3D Base[2]:straight_sol;%{PE}
;FOLD Parameters ;%{h}
;Params IlfProvider=kukaroboter.basistech.inlineforms.movement.spline; Kuka.IsGlobalPoint=False; Kuka.PointName=P322; Kuka.BlendingEnabled=False; Kuka.MoveDataName=CPDAT322; Kuka.VelocityPath=2.000; Kuka.VelocityFieldEnabled=True; Kuka.ColDetectFieldEnabled=True; Kuka.CurrentCDSetIndex=0; Kuka.MovementParameterFieldEnabled=True; IlfCommand=SLIN
;ENDFOLD
SLIN XP322 WITH $VEL = SVEL_CP(2.0, , LCPDAT322),$TOOL = STOOL2(FP322),$BASE = SBASE(FP322.BASE_NO),$IPO_MODE = SIPO_MODE(FP322.IPO_FRAME),$LOAD = SLOAD(FP322.TOOL_NO),$ACC = SACC_CP(LCPDAT322),$ORI_TYPE = SORI_TYP(LCPDAT322),$APO = SAPO(LCPDAT322),$JERK = SJERK(LCPDAT322),$COLLMON_TOL_PRO[1] = USE_CM_PRO_VALUES(0)
;ENDFOLD

;FOLD SLIN P323 Vel=2 m/s CPDAT323 Tool[4]:Microflown3D Base[2]:straight_sol;%{PE}
;FOLD Parameters ;%{h}
;Params IlfProvider=kukaroboter.basistech.inlineforms.movement.spline; Kuka.IsGlobalPoint=False; Kuka.PointName=P323; Kuka.BlendingEnabled=False; Kuka.MoveDataName=CPDAT323; Kuka.VelocityPath=2.000; Kuka.VelocityFieldEnabled=True; Kuka.ColDetectFieldEnabled=True; Kuka.CurrentCDSetIndex=0; Kuka.MovementParameterFieldEnabled=True; IlfCommand=SLIN
;ENDFOLD
SLIN XP323 WITH $VEL = SVEL_CP(2.0, , LCPDAT323),$TOOL = STOOL2(FP323),$BASE = SBASE(FP323.BASE_NO),$IPO_MODE = SIPO_MODE(FP323.IPO_FRAME),$LOAD = SLOAD(FP323.TOOL_NO),$ACC = SACC_CP(LCPDAT323),$ORI_TYPE = SORI_TYP(LCPDAT323),$APO = SAPO(LCPDAT323),$JERK = SJERK(LCPDAT323),$COLLMON_TOL_PRO[1] = USE_CM_PRO_VALUES(0)
;ENDFOLD

;FOLD SLIN P324 Vel=2 m/s CPDAT324 Tool[4]:Microflown3D Base[2]:straight_sol;%{PE}
;FOLD Parameters ;%{h}
;Params IlfProvider=kukaroboter.basistech.inlineforms.movement.spline; Kuka.IsGlobalPoint=False; Kuka.PointName=P324; Kuka.BlendingEnabled=False; Kuka.MoveDataName=CPDAT324; Kuka.VelocityPath=2.000; Kuka.VelocityFieldEnabled=True; Kuka.ColDetectFieldEnabled=True; Kuka.CurrentCDSetIndex=0; Kuka.MovementParameterFieldEnabled=True; IlfCommand=SLIN
;ENDFOLD
SLIN XP324 WITH $VEL = SVEL_CP(2.0, , LCPDAT324),$TOOL = STOOL2(FP324),$BASE = SBASE(FP324.BASE_NO),$IPO_MODE = SIPO_MODE(FP324.IPO_FRAME),$LOAD = SLOAD(FP324.TOOL_NO),$ACC = SACC_CP(LCPDAT324),$ORI_TYPE = SORI_TYP(LCPDAT324),$APO = SAPO(LCPDAT324),$JERK = SJERK(LCPDAT324),$COLLMON_TOL_PRO[1] = USE_CM_PRO_VALUES(0)
;ENDFOLD

;FOLD SLIN P325 Vel=2 m/s CPDAT325 Tool[4]:Microflown3D Base[2]:straight_sol;%{PE}
;FOLD Parameters ;%{h}
;Params IlfProvider=kukaroboter.basistech.inlineforms.movement.spline; Kuka.IsGlobalPoint=False; Kuka.PointName=P325; Kuka.BlendingEnabled=False; Kuka.MoveDataName=CPDAT325; Kuka.VelocityPath=2.000; Kuka.VelocityFieldEnabled=True; Kuka.ColDetectFieldEnabled=True; Kuka.CurrentCDSetIndex=0; Kuka.MovementParameterFieldEnabled=True; IlfCommand=SLIN
;ENDFOLD
SLIN XP325 WITH $VEL = SVEL_CP(2.0, , LCPDAT325),$TOOL = STOOL2(FP325),$BASE = SBASE(FP325.BASE_NO),$IPO_MODE = SIPO_MODE(FP325.IPO_FRAME),$LOAD = SLOAD(FP325.TOOL_NO),$ACC = SACC_CP(LCPDAT325),$ORI_TYPE = SORI_TYP(LCPDAT325),$APO = SAPO(LCPDAT325),$JERK = SJERK(LCPDAT325),$COLLMON_TOL_PRO[1] = USE_CM_PRO_VALUES(0)
;ENDFOLD

;FOLD SLIN P326 Vel=2 m/s CPDAT326 Tool[4]:Microflown3D Base[2]:straight_sol;%{PE}
;FOLD Parameters ;%{h}
;Params IlfProvider=kukaroboter.basistech.inlineforms.movement.spline; Kuka.IsGlobalPoint=False; Kuka.PointName=P326; Kuka.BlendingEnabled=False; Kuka.MoveDataName=CPDAT326; Kuka.VelocityPath=2.000; Kuka.VelocityFieldEnabled=True; Kuka.ColDetectFieldEnabled=True; Kuka.CurrentCDSetIndex=0; Kuka.MovementParameterFieldEnabled=True; IlfCommand=SLIN
;ENDFOLD
SLIN XP326 WITH $VEL = SVEL_CP(2.0, , LCPDAT326),$TOOL = STOOL2(FP326),$BASE = SBASE(FP326.BASE_NO),$IPO_MODE = SIPO_MODE(FP326.IPO_FRAME),$LOAD = SLOAD(FP326.TOOL_NO),$ACC = SACC_CP(LCPDAT326),$ORI_TYPE = SORI_TYP(LCPDAT326),$APO = SAPO(LCPDAT326),$JERK = SJERK(LCPDAT326),$COLLMON_TOL_PRO[1] = USE_CM_PRO_VALUES(0)
;ENDFOLD

;FOLD SLIN P327 Vel=2 m/s CPDAT327 Tool[4]:Microflown3D Base[2]:straight_sol;%{PE}
;FOLD Parameters ;%{h}
;Params IlfProvider=kukaroboter.basistech.inlineforms.movement.spline; Kuka.IsGlobalPoint=False; Kuka.PointName=P327; Kuka.BlendingEnabled=False; Kuka.MoveDataName=CPDAT327; Kuka.VelocityPath=2.000; Kuka.VelocityFieldEnabled=True; Kuka.ColDetectFieldEnabled=True; Kuka.CurrentCDSetIndex=0; Kuka.MovementParameterFieldEnabled=True; IlfCommand=SLIN
;ENDFOLD
SLIN XP327 WITH $VEL = SVEL_CP(2.0, , LCPDAT327),$TOOL = STOOL2(FP327),$BASE = SBASE(FP327.BASE_NO),$IPO_MODE = SIPO_MODE(FP327.IPO_FRAME),$LOAD = SLOAD(FP327.TOOL_NO),$ACC = SACC_CP(LCPDAT327),$ORI_TYPE = SORI_TYP(LCPDAT327),$APO = SAPO(LCPDAT327),$JERK = SJERK(LCPDAT327),$COLLMON_TOL_PRO[1] = USE_CM_PRO_VALUES(0)
;ENDFOLD

;FOLD SLIN P328 Vel=2 m/s CPDAT328 Tool[4]:Microflown3D Base[2]:straight_sol;%{PE}
;FOLD Parameters ;%{h}
;Params IlfProvider=kukaroboter.basistech.inlineforms.movement.spline; Kuka.IsGlobalPoint=False; Kuka.PointName=P328; Kuka.BlendingEnabled=False; Kuka.MoveDataName=CPDAT328; Kuka.VelocityPath=2.000; Kuka.VelocityFieldEnabled=True; Kuka.ColDetectFieldEnabled=True; Kuka.CurrentCDSetIndex=0; Kuka.MovementParameterFieldEnabled=True; IlfCommand=SLIN
;ENDFOLD
SLIN XP328 WITH $VEL = SVEL_CP(2.0, , LCPDAT328),$TOOL = STOOL2(FP328),$BASE = SBASE(FP328.BASE_NO),$IPO_MODE = SIPO_MODE(FP328.IPO_FRAME),$LOAD = SLOAD(FP328.TOOL_NO),$ACC = SACC_CP(LCPDAT328),$ORI_TYPE = SORI_TYP(LCPDAT328),$APO = SAPO(LCPDAT328),$JERK = SJERK(LCPDAT328),$COLLMON_TOL_PRO[1] = USE_CM_PRO_VALUES(0)
;ENDFOLD

;FOLD SLIN P329 Vel=2 m/s CPDAT329 Tool[4]:Microflown3D Base[2]:straight_sol;%{PE}
;FOLD Parameters ;%{h}
;Params IlfProvider=kukaroboter.basistech.inlineforms.movement.spline; Kuka.IsGlobalPoint=False; Kuka.PointName=P329; Kuka.BlendingEnabled=False; Kuka.MoveDataName=CPDAT329; Kuka.VelocityPath=2.000; Kuka.VelocityFieldEnabled=True; Kuka.ColDetectFieldEnabled=True; Kuka.CurrentCDSetIndex=0; Kuka.MovementParameterFieldEnabled=True; IlfCommand=SLIN
;ENDFOLD
SLIN XP329 WITH $VEL = SVEL_CP(2.0, , LCPDAT329),$TOOL = STOOL2(FP329),$BASE = SBASE(FP329.BASE_NO),$IPO_MODE = SIPO_MODE(FP329.IPO_FRAME),$LOAD = SLOAD(FP329.TOOL_NO),$ACC = SACC_CP(LCPDAT329),$ORI_TYPE = SORI_TYP(LCPDAT329),$APO = SAPO(LCPDAT329),$JERK = SJERK(LCPDAT329),$COLLMON_TOL_PRO[1] = USE_CM_PRO_VALUES(0)
;ENDFOLD

;FOLD SLIN P330 Vel=2 m/s CPDAT330 Tool[4]:Microflown3D Base[2]:straight_sol;%{PE}
;FOLD Parameters ;%{h}
;Params IlfProvider=kukaroboter.basistech.inlineforms.movement.spline; Kuka.IsGlobalPoint=False; Kuka.PointName=P330; Kuka.BlendingEnabled=False; Kuka.MoveDataName=CPDAT330; Kuka.VelocityPath=2.000; Kuka.VelocityFieldEnabled=True; Kuka.ColDetectFieldEnabled=True; Kuka.CurrentCDSetIndex=0; Kuka.MovementParameterFieldEnabled=True; IlfCommand=SLIN
;ENDFOLD
SLIN XP330 WITH $VEL = SVEL_CP(2.0, , LCPDAT330),$TOOL = STOOL2(FP330),$BASE = SBASE(FP330.BASE_NO),$IPO_MODE = SIPO_MODE(FP330.IPO_FRAME),$LOAD = SLOAD(FP330.TOOL_NO),$ACC = SACC_CP(LCPDAT330),$ORI_TYPE = SORI_TYP(LCPDAT330),$APO = SAPO(LCPDAT330),$JERK = SJERK(LCPDAT330),$COLLMON_TOL_PRO[1] = USE_CM_PRO_VALUES(0)
;ENDFOLD

;FOLD SLIN P331 Vel=2 m/s CPDAT331 Tool[4]:Microflown3D Base[2]:straight_sol;%{PE}
;FOLD Parameters ;%{h}
;Params IlfProvider=kukaroboter.basistech.inlineforms.movement.spline; Kuka.IsGlobalPoint=False; Kuka.PointName=P331; Kuka.BlendingEnabled=False; Kuka.MoveDataName=CPDAT331; Kuka.VelocityPath=2.000; Kuka.VelocityFieldEnabled=True; Kuka.ColDetectFieldEnabled=True; Kuka.CurrentCDSetIndex=0; Kuka.MovementParameterFieldEnabled=True; IlfCommand=SLIN
;ENDFOLD
SLIN XP331 WITH $VEL = SVEL_CP(2.0, , LCPDAT331),$TOOL = STOOL2(FP331),$BASE = SBASE(FP331.BASE_NO),$IPO_MODE = SIPO_MODE(FP331.IPO_FRAME),$LOAD = SLOAD(FP331.TOOL_NO),$ACC = SACC_CP(LCPDAT331),$ORI_TYPE = SORI_TYP(LCPDAT331),$APO = SAPO(LCPDAT331),$JERK = SJERK(LCPDAT331),$COLLMON_TOL_PRO[1] = USE_CM_PRO_VALUES(0)
;ENDFOLD

;FOLD SLIN P332 Vel=2 m/s CPDAT332 Tool[4]:Microflown3D Base[2]:straight_sol;%{PE}
;FOLD Parameters ;%{h}
;Params IlfProvider=kukaroboter.basistech.inlineforms.movement.spline; Kuka.IsGlobalPoint=False; Kuka.PointName=P332; Kuka.BlendingEnabled=False; Kuka.MoveDataName=CPDAT332; Kuka.VelocityPath=2.000; Kuka.VelocityFieldEnabled=True; Kuka.ColDetectFieldEnabled=True; Kuka.CurrentCDSetIndex=0; Kuka.MovementParameterFieldEnabled=True; IlfCommand=SLIN
;ENDFOLD
SLIN XP332 WITH $VEL = SVEL_CP(2.0, , LCPDAT332),$TOOL = STOOL2(FP332),$BASE = SBASE(FP332.BASE_NO),$IPO_MODE = SIPO_MODE(FP332.IPO_FRAME),$LOAD = SLOAD(FP332.TOOL_NO),$ACC = SACC_CP(LCPDAT332),$ORI_TYPE = SORI_TYP(LCPDAT332),$APO = SAPO(LCPDAT332),$JERK = SJERK(LCPDAT332),$COLLMON_TOL_PRO[1] = USE_CM_PRO_VALUES(0)
;ENDFOLD

;FOLD SLIN P333 Vel=2 m/s CPDAT333 Tool[4]:Microflown3D Base[2]:straight_sol;%{PE}
;FOLD Parameters ;%{h}
;Params IlfProvider=kukaroboter.basistech.inlineforms.movement.spline; Kuka.IsGlobalPoint=False; Kuka.PointName=P333; Kuka.BlendingEnabled=False; Kuka.MoveDataName=CPDAT333; Kuka.VelocityPath=2.000; Kuka.VelocityFieldEnabled=True; Kuka.ColDetectFieldEnabled=True; Kuka.CurrentCDSetIndex=0; Kuka.MovementParameterFieldEnabled=True; IlfCommand=SLIN
;ENDFOLD
SLIN XP333 WITH $VEL = SVEL_CP(2.0, , LCPDAT333),$TOOL = STOOL2(FP333),$BASE = SBASE(FP333.BASE_NO),$IPO_MODE = SIPO_MODE(FP333.IPO_FRAME),$LOAD = SLOAD(FP333.TOOL_NO),$ACC = SACC_CP(LCPDAT333),$ORI_TYPE = SORI_TYP(LCPDAT333),$APO = SAPO(LCPDAT333),$JERK = SJERK(LCPDAT333),$COLLMON_TOL_PRO[1] = USE_CM_PRO_VALUES(0)
;ENDFOLD

;FOLD SLIN P334 Vel=2 m/s CPDAT334 Tool[4]:Microflown3D Base[2]:straight_sol;%{PE}
;FOLD Parameters ;%{h}
;Params IlfProvider=kukaroboter.basistech.inlineforms.movement.spline; Kuka.IsGlobalPoint=False; Kuka.PointName=P334; Kuka.BlendingEnabled=False; Kuka.MoveDataName=CPDAT334; Kuka.VelocityPath=2.000; Kuka.VelocityFieldEnabled=True; Kuka.ColDetectFieldEnabled=True; Kuka.CurrentCDSetIndex=0; Kuka.MovementParameterFieldEnabled=True; IlfCommand=SLIN
;ENDFOLD
SLIN XP334 WITH $VEL = SVEL_CP(2.0, , LCPDAT334),$TOOL = STOOL2(FP334),$BASE = SBASE(FP334.BASE_NO),$IPO_MODE = SIPO_MODE(FP334.IPO_FRAME),$LOAD = SLOAD(FP334.TOOL_NO),$ACC = SACC_CP(LCPDAT334),$ORI_TYPE = SORI_TYP(LCPDAT334),$APO = SAPO(LCPDAT334),$JERK = SJERK(LCPDAT334),$COLLMON_TOL_PRO[1] = USE_CM_PRO_VALUES(0)
;ENDFOLD

;FOLD SLIN P335 Vel=2 m/s CPDAT335 Tool[4]:Microflown3D Base[2]:straight_sol;%{PE}
;FOLD Parameters ;%{h}
;Params IlfProvider=kukaroboter.basistech.inlineforms.movement.spline; Kuka.IsGlobalPoint=False; Kuka.PointName=P335; Kuka.BlendingEnabled=False; Kuka.MoveDataName=CPDAT335; Kuka.VelocityPath=2.000; Kuka.VelocityFieldEnabled=True; Kuka.ColDetectFieldEnabled=True; Kuka.CurrentCDSetIndex=0; Kuka.MovementParameterFieldEnabled=True; IlfCommand=SLIN
;ENDFOLD
SLIN XP335 WITH $VEL = SVEL_CP(2.0, , LCPDAT335),$TOOL = STOOL2(FP335),$BASE = SBASE(FP335.BASE_NO),$IPO_MODE = SIPO_MODE(FP335.IPO_FRAME),$LOAD = SLOAD(FP335.TOOL_NO),$ACC = SACC_CP(LCPDAT335),$ORI_TYPE = SORI_TYP(LCPDAT335),$APO = SAPO(LCPDAT335),$JERK = SJERK(LCPDAT335),$COLLMON_TOL_PRO[1] = USE_CM_PRO_VALUES(0)
;ENDFOLD

;FOLD SLIN P336 Vel=2 m/s CPDAT336 Tool[4]:Microflown3D Base[2]:straight_sol;%{PE}
;FOLD Parameters ;%{h}
;Params IlfProvider=kukaroboter.basistech.inlineforms.movement.spline; Kuka.IsGlobalPoint=False; Kuka.PointName=P336; Kuka.BlendingEnabled=False; Kuka.MoveDataName=CPDAT336; Kuka.VelocityPath=2.000; Kuka.VelocityFieldEnabled=True; Kuka.ColDetectFieldEnabled=True; Kuka.CurrentCDSetIndex=0; Kuka.MovementParameterFieldEnabled=True; IlfCommand=SLIN
;ENDFOLD
SLIN XP336 WITH $VEL = SVEL_CP(2.0, , LCPDAT336),$TOOL = STOOL2(FP336),$BASE = SBASE(FP336.BASE_NO),$IPO_MODE = SIPO_MODE(FP336.IPO_FRAME),$LOAD = SLOAD(FP336.TOOL_NO),$ACC = SACC_CP(LCPDAT336),$ORI_TYPE = SORI_TYP(LCPDAT336),$APO = SAPO(LCPDAT336),$JERK = SJERK(LCPDAT336),$COLLMON_TOL_PRO[1] = USE_CM_PRO_VALUES(0)
;ENDFOLD

;FOLD SLIN P337 Vel=2 m/s CPDAT337 Tool[4]:Microflown3D Base[2]:straight_sol;%{PE}
;FOLD Parameters ;%{h}
;Params IlfProvider=kukaroboter.basistech.inlineforms.movement.spline; Kuka.IsGlobalPoint=False; Kuka.PointName=P337; Kuka.BlendingEnabled=False; Kuka.MoveDataName=CPDAT337; Kuka.VelocityPath=2.000; Kuka.VelocityFieldEnabled=True; Kuka.ColDetectFieldEnabled=True; Kuka.CurrentCDSetIndex=0; Kuka.MovementParameterFieldEnabled=True; IlfCommand=SLIN
;ENDFOLD
SLIN XP337 WITH $VEL = SVEL_CP(2.0, , LCPDAT337),$TOOL = STOOL2(FP337),$BASE = SBASE(FP337.BASE_NO),$IPO_MODE = SIPO_MODE(FP337.IPO_FRAME),$LOAD = SLOAD(FP337.TOOL_NO),$ACC = SACC_CP(LCPDAT337),$ORI_TYPE = SORI_TYP(LCPDAT337),$APO = SAPO(LCPDAT337),$JERK = SJERK(LCPDAT337),$COLLMON_TOL_PRO[1] = USE_CM_PRO_VALUES(0)
;ENDFOLD

;FOLD SLIN P338 Vel=2 m/s CPDAT338 Tool[4]:Microflown3D Base[2]:straight_sol;%{PE}
;FOLD Parameters ;%{h}
;Params IlfProvider=kukaroboter.basistech.inlineforms.movement.spline; Kuka.IsGlobalPoint=False; Kuka.PointName=P338; Kuka.BlendingEnabled=False; Kuka.MoveDataName=CPDAT338; Kuka.VelocityPath=2.000; Kuka.VelocityFieldEnabled=True; Kuka.ColDetectFieldEnabled=True; Kuka.CurrentCDSetIndex=0; Kuka.MovementParameterFieldEnabled=True; IlfCommand=SLIN
;ENDFOLD
SLIN XP338 WITH $VEL = SVEL_CP(2.0, , LCPDAT338),$TOOL = STOOL2(FP338),$BASE = SBASE(FP338.BASE_NO),$IPO_MODE = SIPO_MODE(FP338.IPO_FRAME),$LOAD = SLOAD(FP338.TOOL_NO),$ACC = SACC_CP(LCPDAT338),$ORI_TYPE = SORI_TYP(LCPDAT338),$APO = SAPO(LCPDAT338),$JERK = SJERK(LCPDAT338),$COLLMON_TOL_PRO[1] = USE_CM_PRO_VALUES(0)
;ENDFOLD

;FOLD SLIN P339 Vel=2 m/s CPDAT339 Tool[4]:Microflown3D Base[2]:straight_sol;%{PE}
;FOLD Parameters ;%{h}
;Params IlfProvider=kukaroboter.basistech.inlineforms.movement.spline; Kuka.IsGlobalPoint=False; Kuka.PointName=P339; Kuka.BlendingEnabled=False; Kuka.MoveDataName=CPDAT339; Kuka.VelocityPath=2.000; Kuka.VelocityFieldEnabled=True; Kuka.ColDetectFieldEnabled=True; Kuka.CurrentCDSetIndex=0; Kuka.MovementParameterFieldEnabled=True; IlfCommand=SLIN
;ENDFOLD
SLIN XP339 WITH $VEL = SVEL_CP(2.0, , LCPDAT339),$TOOL = STOOL2(FP339),$BASE = SBASE(FP339.BASE_NO),$IPO_MODE = SIPO_MODE(FP339.IPO_FRAME),$LOAD = SLOAD(FP339.TOOL_NO),$ACC = SACC_CP(LCPDAT339),$ORI_TYPE = SORI_TYP(LCPDAT339),$APO = SAPO(LCPDAT339),$JERK = SJERK(LCPDAT339),$COLLMON_TOL_PRO[1] = USE_CM_PRO_VALUES(0)
;ENDFOLD

;FOLD SLIN P340 Vel=2 m/s CPDAT340 Tool[4]:Microflown3D Base[2]:straight_sol;%{PE}
;FOLD Parameters ;%{h}
;Params IlfProvider=kukaroboter.basistech.inlineforms.movement.spline; Kuka.IsGlobalPoint=False; Kuka.PointName=P340; Kuka.BlendingEnabled=False; Kuka.MoveDataName=CPDAT340; Kuka.VelocityPath=2.000; Kuka.VelocityFieldEnabled=True; Kuka.ColDetectFieldEnabled=True; Kuka.CurrentCDSetIndex=0; Kuka.MovementParameterFieldEnabled=True; IlfCommand=SLIN
;ENDFOLD
SLIN XP340 WITH $VEL = SVEL_CP(2.0, , LCPDAT340),$TOOL = STOOL2(FP340),$BASE = SBASE(FP340.BASE_NO),$IPO_MODE = SIPO_MODE(FP340.IPO_FRAME),$LOAD = SLOAD(FP340.TOOL_NO),$ACC = SACC_CP(LCPDAT340),$ORI_TYPE = SORI_TYP(LCPDAT340),$APO = SAPO(LCPDAT340),$JERK = SJERK(LCPDAT340),$COLLMON_TOL_PRO[1] = USE_CM_PRO_VALUES(0)
;ENDFOLD

;FOLD SLIN P341 Vel=2 m/s CPDAT341 Tool[4]:Microflown3D Base[2]:straight_sol;%{PE}
;FOLD Parameters ;%{h}
;Params IlfProvider=kukaroboter.basistech.inlineforms.movement.spline; Kuka.IsGlobalPoint=False; Kuka.PointName=P341; Kuka.BlendingEnabled=False; Kuka.MoveDataName=CPDAT341; Kuka.VelocityPath=2.000; Kuka.VelocityFieldEnabled=True; Kuka.ColDetectFieldEnabled=True; Kuka.CurrentCDSetIndex=0; Kuka.MovementParameterFieldEnabled=True; IlfCommand=SLIN
;ENDFOLD
SLIN XP341 WITH $VEL = SVEL_CP(2.0, , LCPDAT341),$TOOL = STOOL2(FP341),$BASE = SBASE(FP341.BASE_NO),$IPO_MODE = SIPO_MODE(FP341.IPO_FRAME),$LOAD = SLOAD(FP341.TOOL_NO),$ACC = SACC_CP(LCPDAT341),$ORI_TYPE = SORI_TYP(LCPDAT341),$APO = SAPO(LCPDAT341),$JERK = SJERK(LCPDAT341),$COLLMON_TOL_PRO[1] = USE_CM_PRO_VALUES(0)
;ENDFOLD

;FOLD SLIN P342 Vel=2 m/s CPDAT342 Tool[4]:Microflown3D Base[2]:straight_sol;%{PE}
;FOLD Parameters ;%{h}
;Params IlfProvider=kukaroboter.basistech.inlineforms.movement.spline; Kuka.IsGlobalPoint=False; Kuka.PointName=P342; Kuka.BlendingEnabled=False; Kuka.MoveDataName=CPDAT342; Kuka.VelocityPath=2.000; Kuka.VelocityFieldEnabled=True; Kuka.ColDetectFieldEnabled=True; Kuka.CurrentCDSetIndex=0; Kuka.MovementParameterFieldEnabled=True; IlfCommand=SLIN
;ENDFOLD
SLIN XP342 WITH $VEL = SVEL_CP(2.0, , LCPDAT342),$TOOL = STOOL2(FP342),$BASE = SBASE(FP342.BASE_NO),$IPO_MODE = SIPO_MODE(FP342.IPO_FRAME),$LOAD = SLOAD(FP342.TOOL_NO),$ACC = SACC_CP(LCPDAT342),$ORI_TYPE = SORI_TYP(LCPDAT342),$APO = SAPO(LCPDAT342),$JERK = SJERK(LCPDAT342),$COLLMON_TOL_PRO[1] = USE_CM_PRO_VALUES(0)
;ENDFOLD

;FOLD SLIN P343 Vel=2 m/s CPDAT343 Tool[4]:Microflown3D Base[2]:straight_sol;%{PE}
;FOLD Parameters ;%{h}
;Params IlfProvider=kukaroboter.basistech.inlineforms.movement.spline; Kuka.IsGlobalPoint=False; Kuka.PointName=P343; Kuka.BlendingEnabled=False; Kuka.MoveDataName=CPDAT343; Kuka.VelocityPath=2.000; Kuka.VelocityFieldEnabled=True; Kuka.ColDetectFieldEnabled=True; Kuka.CurrentCDSetIndex=0; Kuka.MovementParameterFieldEnabled=True; IlfCommand=SLIN
;ENDFOLD
SLIN XP343 WITH $VEL = SVEL_CP(2.0, , LCPDAT343),$TOOL = STOOL2(FP343),$BASE = SBASE(FP343.BASE_NO),$IPO_MODE = SIPO_MODE(FP343.IPO_FRAME),$LOAD = SLOAD(FP343.TOOL_NO),$ACC = SACC_CP(LCPDAT343),$ORI_TYPE = SORI_TYP(LCPDAT343),$APO = SAPO(LCPDAT343),$JERK = SJERK(LCPDAT343),$COLLMON_TOL_PRO[1] = USE_CM_PRO_VALUES(0)
;ENDFOLD

;FOLD SLIN P344 Vel=2 m/s CPDAT344 Tool[4]:Microflown3D Base[2]:straight_sol;%{PE}
;FOLD Parameters ;%{h}
;Params IlfProvider=kukaroboter.basistech.inlineforms.movement.spline; Kuka.IsGlobalPoint=False; Kuka.PointName=P344; Kuka.BlendingEnabled=False; Kuka.MoveDataName=CPDAT344; Kuka.VelocityPath=2.000; Kuka.VelocityFieldEnabled=True; Kuka.ColDetectFieldEnabled=True; Kuka.CurrentCDSetIndex=0; Kuka.MovementParameterFieldEnabled=True; IlfCommand=SLIN
;ENDFOLD
SLIN XP344 WITH $VEL = SVEL_CP(2.0, , LCPDAT344),$TOOL = STOOL2(FP344),$BASE = SBASE(FP344.BASE_NO),$IPO_MODE = SIPO_MODE(FP344.IPO_FRAME),$LOAD = SLOAD(FP344.TOOL_NO),$ACC = SACC_CP(LCPDAT344),$ORI_TYPE = SORI_TYP(LCPDAT344),$APO = SAPO(LCPDAT344),$JERK = SJERK(LCPDAT344),$COLLMON_TOL_PRO[1] = USE_CM_PRO_VALUES(0)
;ENDFOLD

;FOLD SPTP HOME Vel=100 % DEFAULT ;%{PE}
;FOLD Parameters ;%{h}
;Params IlfProvider=kukaroboter.basistech.inlineforms.movement.spline; Kuka.IsGlobalPoint=False; Kuka.PointName=HOME; Kuka.BlendingEnabled=False; Kuka.MoveDataPtpName=DEFAULT; Kuka.VelocityPtp=100; Kuka.VelocityFieldEnabled=True; Kuka.CurrentCDSetIndex=0; Kuka.MovementParameterFieldEnabled=True; IlfCommand=SPTP
;ENDFOLD
SPTP XHOME WITH $VEL_AXIS[1] = SVEL_JOINT(100.0), $TOOL = STOOL2(FHOME), $BASE = SBASE(FHOME.BASE_NO), $IPO_MODE = SIPO_MODE(FHOME.IPO_FRAME), $LOAD = SLOAD(FHOME.TOOL_NO), $ACC_AXIS[1] = SACC_JOINT(PDEFAULT), $APO = SAPO_PTP(PDEFAULT), $GEAR_JERK[1] = SGEAR_JERK(PDEFAULT), $COLLMON_TOL_PRO[1] = USE_CM_PRO_VALUES(0)
;ENDFOLD

END

--- near_field234.dat ---
&ACCESS RVP
&REL 344
&PARAM EDITMASK = *
&PARAM TEMPLATE = C:\KRC\Roboter\Template\vorgabe
&PARAM DISKPATH = KRC:\R1\Parcours\Nicolas F
DEFDAT parcour-time07_01_50-date05_29_2022
;FOLD EXTERNAL DECLARATIONS;%{PE}%MKUKATPBASIS,%CEXT,%VCOMMON,%P
;FOLD BASISTECH EXT;%{PE}%MKUKATPBASIS,%CEXT,%VEXT,%P
EXT  BAS (BAS_COMMAND  :IN,REAL  :IN )
DECL INT SUCCESS
;ENDFOLD (BASISTECH EXT)
;FOLD USER EXT;%{E}%MKUKATPUSER,%CEXT,%VEXT,%P
;Make your modifications here

;ENDFOLD (USER EXT)
;ENDFOLD (EXTERNAL DECLARATIONS)

DECL MODULEPARAM_T LAST_TP_PARAMS={PARAMS[] "Kuka.VelocityFieldEnabled=False; Kuka.ColDetectFieldEnabled=False; Kuka.MovementParameterFieldEnabled=False; Kuka.IsAngleEnabled=False; Kuka.PointName=P1; Kuka.FrameData.base_no=2; Kuka.FrameData.tool_no=4; Kuka.FrameData.ipo_frame=#BASE; Kuka.isglobalpoint=False; Kuka.MoveDataPtpName=PDAT1; Kuka.MovementDataPdat.apo_mode=#CDIS; Kuka.MovementDataPdat.apo_dist=500; Kuka.MovementData.vel=75; Kuka.MovementData.acc=100; Kuka.MovementData.exax_ign=0; Kuka.VelocityPtp=75; Kuka.BlendingEnabled=False; Kuka.APXEnabled=False; Kuka.CurrentCDSetIndex=0"}

DECL E6POS XP1={X 0,Y 0,Z 800,A 0,B -90,C 180,S 6,T 50,E1 0.0,E2 0.0,E3 0.0,E4 0.0,E5 0.0,E6 0.0}
DECL FDAT FP1={TOOL_NO 4,BASE_NO 2,IPO_FRAME #BASE,POINT2[] " "}
DECL PDAT PPDAT1={VEL 75.000,ACC 100.000,APO_DIST 500.000,APO_MODE #CDIS,GEAR_JERK 100.000,EXAX_IGN 0}

DECL E6POS XP2={X -263.5,Y 0,Z 800,A 0,B -45,C 180,S 6,T 16,E1 0.0,E2 0.0,E3 0.0,E4 0.0,E5 0.0,E6 0.0}
DECL FDAT FP2={TOOL_NO 4,BASE_NO 2,IPO_FRAME #BASE,POINT2[] " "}
DECL LDAT LCPDAT2={VEL 1,ACC 100.000,APO_DIST 500.000,APO_FAC 50.0000,AXIS_VEL 100.000,AXIS_ACC 100.000,ORI_TYP #VAR,CIRC_TYP #BASE,JERK_FAC 50.0000,GEAR_JERK 100.000,EXAX_IGN 0}

DECL E6POS XP3={X -233.5,Y -233.5,Z 0,A 0,B -45,C 180,S 6,T 16,E1 0.0,E2 0.0,E3 0.0,E4 0.0,E5 0.0,E6 0.0}
DECL FDAT FP3={TOOL_NO 4,BASE_NO 2,IPO_FRAME #BASE,POINT2[] " "}
DECL LDAT LCPDAT3={VEL 2,ACC 100.000,APO_DIST 500.000,APO_FAC 50.0000,AXIS_VEL 100.000,AXIS_ACC 100.000,ORI_TYP #VAR,CIRC_TYP #BASE,JERK_FAC 50.0000,GEAR_JERK 100.000,EXAX_IGN 0}

DECL E6POS XP4={X -233.5,Y -193.5,Z 0,A 0,B -45,C 180,S 6,T 16,E1 0.0,E2 0.0,E3 0.0,E4 0.0,E5 0.0,E6 0.0}
DECL FDAT FP4={TOOL_NO 4,BASE_NO 2,IPO_FRAME #BASE,POINT2[] " "}
DECL LDAT LCPDAT4={VEL 2,ACC 100.000,APO_DIST 500.000,APO_FAC 50.0000,AXIS_VEL 100.000,AXIS_ACC 100.000,ORI_TYP #VAR,CIRC_TYP #BASE,JERK_FAC 50.0000,GEAR_JERK 100.000,EXAX_IGN 0}

DECL E6POS XP5={X -233.5,Y -153.5,Z 0,A 0,B -45,C 180,S 6,T 16,E1 0.0,E2 0.0,E3 0.0,E4 0.0,E5 0.0,E6 0.0}
DECL FDAT FP5={TOOL_NO 4,BASE_NO 2,IPO_FRAME #BASE,POINT2[] " "}
DECL LDAT LCPDAT5={VEL 2,ACC 100.000,APO_DIST 500.000,APO_FAC 50.0000,AXIS_VEL 100.000,AXIS_ACC 100.000,ORI_TYP #VAR,CIRC_TYP #BASE,JERK_FAC 50.0000,GEAR_JERK 100.000,EXAX_IGN 0}

DECL E6POS XP6={X -233.5,Y -113.5,Z 0,A 0,B -45,C 180,S 6,T 16,E1 0.0,E2 0.0,E3 0.0,E4 0.0,E5 0.0,E6 0.0}
DECL FDAT FP6={TOOL_NO 4,BASE_NO 2,IPO_FRAME #BASE,POINT2[] " "}
DECL LDAT LCPDAT6={VEL 2,ACC 100.000,APO_DIST 500.000,APO_FAC 50.0000,AXIS_VEL 100.000,AXIS_ACC 100.000,ORI_TYP #VAR,CIRC_TYP #BASE,JERK_FAC 50.0000,GEAR_JERK 100.000,EXAX_IGN 0}

DECL E6POS XP7={X -233.5,Y -73.5,Z 0,A 0,B -45,C 180,S 6,T 16,E1 0.0,E2 0.0,E3 0.0,E4 0.0,E5 0.0,E6 0.0}
DECL FDAT FP7={TOOL_NO 4,BASE_NO 2,IPO_FRAME #BASE,POINT2[] " "}
DECL LDAT LCPDAT7={VEL 2,ACC 100.000,APO_DIST 500.000,APO_FAC 50.0000,AXIS_VEL 100.000,AXIS_ACC 100.000,ORI_TYP #VAR,CIRC_TYP #BASE,JERK_FAC 50.0000,GEAR_JERK 100.000,EXAX_IGN 0}

DECL E6POS XP8={X -233.5,Y -33.5,Z 0,A 0,B -45,C 180,S 6,T 16,E1 0.0,E2 0.0,E3 0.0,E4 0.0,E5 0.0,E6 0.0}
DECL FDAT FP8={TOOL_NO 4,BASE_NO 2,IPO_FRAME #BASE,POINT2[] " "}
DECL LDAT LCPDAT8={VEL 2,ACC 100.000,APO_DIST 500.000,APO_FAC 50.0000,AXIS_VEL 100.000,AXIS_ACC 100.000,ORI_TYP #VAR,CIRC_TYP #BASE,JERK_FAC 50.0000,GEAR_JERK 100.000,EXAX_IGN 0}

DECL E6POS XP9={X -233.5,Y 6.5,Z 0,A 0,B -45,C 180,S 6,T 16,E1 0.0,E2 0.0,E3 0.0,E4 0.0,E5 0.0,E6 0.0}
DECL FDAT FP9={TOOL_NO 4,BASE_NO 2,IPO_FRAME #BASE,POINT2[] " "}
DECL LDAT LCPDAT9={VEL 2,ACC 100.000,APO_DIST 500.000,APO_FAC 50.0000,AXIS_VEL 100.000,AXIS_ACC 100.000,ORI_TYP #VAR,CIRC_TYP #BASE,JERK_FAC 50.0000,GEAR_JERK 100.000,EXAX_IGN 0}

DECL E6POS XP10={X -233.5,Y 46.5,Z 0,A 0,B -45,C 180,S 6,T 16,E1 0.0,E2 0.0,E3 0.0,E4 0.0,E5 0.0,E6 0.0}
DECL FDAT FP10={TOOL_NO 4,BASE_NO 2,IPO_FRAME #BASE,POINT2[] " "}
DECL LDAT LCPDAT10={VEL 2,ACC 100.000,APO_DIST 500.000,APO_FAC 50.0000,AXIS_VEL 100.000,AXIS_ACC 100.000,ORI_TYP #VAR,CIRC_TYP #BASE,JERK_FAC 50.0000,GEAR_JERK 100.000,EXAX_IGN 0}

DECL E6POS XP11={X -233.5,Y 86.5,Z 0,A 0,B -45,C 180,S 6,T 16,E1 0.0,E2 0.0,E3 0.0,E4 0.0,E5 0.0,E6 0.0}
DECL FDAT FP11={TOOL_NO 4,BASE_NO 2,IPO_FRAME #BASE,POINT2[] " "}
DECL LDAT LCPDAT11={VEL 2,ACC 100.000,APO_DIST 500.000,APO_FAC 50.0000,AXIS_VEL 100.000,AXIS_ACC 100.000,ORI_TYP #VAR,CIRC_TYP #BASE,JERK_FAC 50.0000,GEAR_JERK 100.000,EXAX_IGN 0}

DECL E6POS XP12={X -233.5,Y 126.5,Z 0,A 0,B -45,C 180,S 6,T 16,E1 0.0,E2 0.0,E3 0.0,E4 0.0,E5 0.0,E6 0.0}
DECL FDAT FP12={TOOL_NO 4,BASE_NO 2,IPO_FRAME #BASE,POINT2[] " "}
DECL LDAT LCPDAT12={VEL 2,ACC 100.000,APO_DIST 500.000,APO_FAC 50.0000,AXIS_VEL 100.000,AXIS_ACC 100.000,ORI_TYP #VAR,CIRC_TYP #BASE,JERK_FAC 50.0000,GEAR_JERK 100.000,EXAX_IGN 0}

DECL E6POS XP13={X -233.5,Y 166.5,Z 0,A 0,B -45,C 180,S 6,T 16,E1 0.0,E2 0.0,E3 0.0,E4 0.0,E5 0.0,E6 0.0}
DECL FDAT FP13={TOOL_NO 4,BASE_NO 2,IPO_FRAME #BASE,POINT2[] " "}
DECL LDAT LCPDAT13={VEL 2,ACC 100.000,APO_DIST 500.000,APO_FAC 50.0000,AXIS_VEL 100.000,AXIS_ACC 100.000,ORI_TYP #VAR,CIRC_TYP #BASE,JERK_FAC 50.0000,GEAR_JERK 100.000,EXAX_IGN 0}

DECL E6POS XP14={X -233.5,Y 206.5,Z 0,A 0,B -45,C 180,S 6,T 16,E1 0.0,E2 0.0,E3 0.0,E4 0.0,E5 0.0,E6 0.0}
DECL FDAT FP14={TOOL_NO 4,BASE_NO 2,IPO_FRAME #BASE,POINT2[] " "}
DECL LDAT LCPDAT14={VEL 2,ACC 100.000,APO_DIST 500.000,APO_FAC 50.0000,AXIS_VEL 100.000,AXIS_ACC 100.000,ORI_TYP #VAR,CIRC_TYP #BASE,JERK_FAC 50.0000,GEAR_JERK 100.000,EXAX_IGN 0}

DECL E6POS XP15={X -233.5,Y 206.5,Z 40,A 0,B -45,C 180,S 6,T 16,E1 0.0,E2 0.0,E3 0.0,E4 0.0,E5 0.0,E6 0.0}
DECL FDAT FP15={TOOL_NO 4,BASE_NO 2,IPO_FRAME #BASE,POINT2[] " "}
DECL LDAT LCPDAT15={VEL 2,ACC 100.000,APO_DIST 500.000,APO_FAC 50.0000,AXIS_VEL 100.000,AXIS_ACC 100.000,ORI_TYP #VAR,CIRC_TYP #BASE,JERK_FAC 50.0000,GEAR_JERK 100.000,EXAX_IGN 0}

DECL E6POS XP16={X -233.5,Y 166.5,Z 40,A 0,B -45,C 180,S 6,T 16,E1 0.0,E2 0.0,E3 0.0,E4 0.0,E5 0.0,E6 0.0}
DECL FDAT FP16={TOOL_NO 4,BASE_NO 2,IPO_FRAME #BASE,POINT2[] " "}
DECL LDAT LCPDAT16={VEL 2,ACC 100.000,APO_DIST 500.000,APO_FAC 50.0000,AXIS_VEL 100.000,AXIS_ACC 100.000,ORI_TYP #VAR,CIRC_TYP #BASE,JERK_FAC 50.0000,GEAR_JERK 100.000,EXAX_IGN 0}

DECL E6POS XP17={X -233.5,Y 126.5,Z 40,A 0,B -45,C 180,S 6,T 16,E1 0.0,E2 0.0,E3 0.0,E4 0.0,E5 0.0,E6 0.0}
DECL FDAT FP17={TOOL_NO 4,BASE_NO 2,IPO_FRAME #BASE,POINT2[] " "}
DECL LDAT LCPDAT17={VEL 2,ACC 100.000,APO_DIST 500.000,APO_FAC 50.0000,AXIS_VEL 100.000,AXIS_ACC 100.000,ORI_TYP #VAR,CIRC_TYP #BASE,JERK_FAC 50.0000,GEAR_JERK 100.000,EXAX_IGN 0}

DECL E6POS XP18={X -233.5,Y 86.5,Z 40,A 0,B -45,C 180,S 6,T 16,E1 0.0,E2 0.0,E3 0.0,E4 0.0,E5 0.0,E6 0.0}
DECL FDAT FP18={TOOL_NO 4,BASE_NO 2,IPO_FRAME #BASE,POINT2[] " "}
DECL LDAT LCPDAT18={VEL 2,ACC 100.000,APO_DIST 500.000,APO_FAC 50.0000,AXIS_VEL 100.000,AXIS_ACC 100.000,ORI_TYP #VAR,CIRC_TYP #BASE,JERK_FAC 50.0000,GEAR_JERK 100.000,EXAX_IGN 0}

DECL E6POS XP19={X -233.5,Y 46.5,Z 40,A 0,B -45,C 180,S 6,T 16,E1 0.0,E2 0.0,E3 0.0,E4 0.0,E5 0.0,E6 0.0}
DECL FDAT FP19={TOOL_NO 4,BASE_NO 2,IPO_FRAME #BASE,POINT2[] " "}
DECL LDAT LCPDAT19={VEL 2,ACC 100.000,APO_DIST 500.000,APO_FAC 50.0000,AXIS_VEL 100.000,AXIS_ACC 100.000,ORI_TYP #VAR,CIRC_TYP #BASE,JERK_FAC 50.0000,GEAR_JERK 100.000,EXAX_IGN 0}

DECL E6POS XP20={X -233.5,Y 6.5,Z 40,A 0,B -45,C 180,S 6,T 16,E1 0.0,E2 0.0,E3 0.0,E4 0.0,E5 0.0,E6 0.0}
DECL FDAT FP20={TOOL_NO 4,BASE_NO 2,IPO_FRAME #BASE,POINT2[] " "}
DECL LDAT LCPDAT20={VEL 2,ACC 100.000,APO_DIST 500.000,APO_FAC 50.0000,AXIS_VEL 100.000,AXIS_ACC 100.000,ORI_TYP #VAR,CIRC_TYP #BASE,JERK_FAC 50.0000,GEAR_JERK 100.000,EXAX_IGN 0}

DECL E6POS XP21={X -233.5,Y -33.5,Z 40,A 0,B -45,C 180,S 6,T 16,E1 0.0,E2 0.0,E3 0.0,E4 0.0,E5 0.0,E6 0.0}
DECL FDAT FP21={TOOL_NO 4,BASE_NO 2,IPO_FRAME #BASE,POINT2[] " "}
DECL LDAT LCPDAT21={VEL 2,ACC 100.000,APO_DIST 500.000,APO_FAC 50.0000,AXIS_VEL 100.000,AXIS_ACC 100.000,ORI_TYP #VAR,CIRC_TYP #BASE,JERK_FAC 50.0000,GEAR_JERK 100.000,EXAX_IGN 0}

DECL E6POS XP22={X -233.5,Y -73.5,Z 40,A 0,B -45,C 180,S 6,T 16,E1 0.0,E2 0.0,E3 0.0,E4 0.0,E5 0.0,E6 0.0}
DECL FDAT FP22={TOOL_NO 4,BASE_NO 2,IPO_FRAME #BASE,POINT2[] " "}
DECL LDAT LCPDAT22={VEL 2,ACC 100.000,APO_DIST 500.000,APO_FAC 50.0000,AXIS_VEL 100.000,AXIS_ACC 100.000,ORI_TYP #VAR,CIRC_TYP #BASE,JERK_FAC 50.0000,GEAR_JERK 100.000,EXAX_IGN 0}

DECL E6POS XP23={X -233.5,Y -113.5,Z 40,A 0,B -45,C 180,S 6,T 16,E1 0.0,E2 0.0,E3 0.0,E4 0.0,E5 0.0,E6 0.0}
DECL FDAT FP23={TOOL_NO 4,BASE_NO 2,IPO_FRAME #BASE,POINT2[] " "}
DECL LDAT LCPDAT23={VEL 2,ACC 100.000,APO_DIST 500.000,APO_FAC 50.0000,AXIS_VEL 100.000,AXIS_ACC 100.000,ORI_TYP #VAR,CIRC_TYP #BASE,JERK_FAC 50.0000,GEAR_JERK 100.000,EXAX_IGN 0}

DECL E6POS XP24={X -233.5,Y -153.5,Z 40,A 0,B -45,C 180,S 6,T 16,E1 0.0,E2 0.0,E3 0.0,E4 0.0,E5 0.0,E6 0.0}
DECL FDAT FP24={TOOL_NO 4,BASE_NO 2,IPO_FRAME #BASE,POINT2[] " "}
DECL LDAT LCPDAT24={VEL 2,ACC 100.000,APO_DIST 500.000,APO_FAC 50.0000,AXIS_VEL 100.000,AXIS_ACC 100.000,ORI_TYP #VAR,CIRC_TYP #BASE,JERK_FAC 50.0000,GEAR_JERK 100.000,EXAX_IGN 0}

DECL E6POS XP25={X -233.5,Y -193.5,Z 40,A 0,B -45,C 180,S 6,T 16,E1 0.0,E2 0.0,E3 0.0,E4 0.0,E5 0.0,E6 0.0}
DECL FDAT FP25={TOOL_NO 4,BASE_NO 2,IPO_FRAME #BASE,POINT2[] " "}
DECL LDAT LCPDAT25={VEL 2,ACC 100.000,APO_DIST 500.000,APO_FAC 50.0000,AXIS_VEL 100.000,AXIS_ACC 100.000,ORI_TYP #VAR,CIRC_TYP #BASE,JERK_FAC 50.0000,GEAR_JERK 100.000,EXAX_IGN 0}

DECL E6POS XP26={X -233.5,Y -233.5,Z 40,A 0,B -45,C 180,S 6,T 16,E1 0.0,E2 0.0,E3 0.0,E4 0.0,E5 0.0,E6 0.0}
DECL FDAT FP26={TOOL_NO 4,BASE_NO 2,IPO_FRAME #BASE,POINT2[] " "}
DECL LDAT LCPDAT26={VEL 2,ACC 100.000,APO_DIST 500.000,APO_FAC 50.0000,AXIS_VEL 100.000,AXIS_ACC 100.000,ORI_TYP #VAR,CIRC_TYP #BASE,JERK_FAC 50.0000,GEAR_JERK 100.000,EXAX_IGN 0}

DECL E6POS XP27={X -233.5,Y -233.5,Z 80,A 0,B -45,C 180,S 6,T 16,E1 0.0,E2 0.0,E3 0.0,E4 0.0,E5 0.0,E6 0.0}
DECL FDAT FP27={TOOL_NO 4,BASE_NO 2,IPO_FRAME #BASE,POINT2[] " "}
DECL LDAT LCPDAT27={VEL 2,ACC 100.000,APO_DIST 500.000,APO_FAC 50.0000,AXIS_VEL 100.000,AXIS_ACC 100.000,ORI_TYP #VAR,CIRC_TYP #BASE,JERK_FAC 50.0000,GEAR_JERK 100.000,EXAX_IGN 0}

DECL E6POS XP28={X -233.5,Y -193.5,Z 80,A 0,B -45,C 180,S 6,T 16,E1 0.0,E2 0.0,E3 0.0,E4 0.0,E5 0.0,E6 0.0}
DECL FDAT FP28={TOOL_NO 4,BASE_NO 2,IPO_FRAME #BASE,POINT2[] " "}
DECL LDAT LCPDAT28={VEL 2,ACC 100.000,APO_DIST 500.000,APO_FAC 50.0000,AXIS_VEL 100.000,AXIS_ACC 100.000,ORI_TYP #VAR,CIRC_TYP #BASE,JERK_FAC 50.0000,GEAR_JERK 100.000,EXAX_IGN 0}

DECL E6POS XP29={X -233.5,Y -153.5,Z 80,A 0,B -45,C 180,S 6,T 16,E1 0.0,E2 0.0,E3 0.0,E4 0.0,E5 0.0,E6 0.0}
DECL FDAT FP29={TOOL_NO 4,BASE_NO 2,IPO_FRAME #BASE,POINT2[] " "}
DECL LDAT LCPDAT29={VEL 2,ACC 100.000,APO_DIST 500.000,APO_FAC 50.0000,AXIS_VEL 100.000,AXIS_ACC 100.000,ORI_TYP #VAR,CIRC_TYP #BASE,JERK_FAC 50.0000,GEAR_JERK 100.000,EXAX_IGN 0}

DECL E6POS XP30={X -233.5,Y -113.5,Z 80,A 0,B -45,C 180,S 6,T 16,E1 0.0,E2 0.0,E3 0.0,E4 0.0,E5 0.0,E6 0.0}
DECL FDAT FP30={TOOL_NO 4,BASE_NO 2,IPO_FRAME #BASE,POINT2[] " "}
DECL LDAT LCPDAT30={VEL 2,ACC 100.000,APO_DIST 500.000,APO_FAC 50.0000,AXIS_VEL 100.000,AXIS_ACC 100.000,ORI_TYP #VAR,CIRC_TYP #BASE,JERK_FAC 50.0000,GEAR_JERK 100.000,EXAX_IGN 0}

DECL E6POS XP31={X -233.5,Y -73.5,Z 80,A 0,B -45,C 180,S 6,T 16,E1 0.0,E2 0.0,E3 0.0,E4 0.0,E5 0.0,E6 0.0}
DECL FDAT FP31={TOOL_NO 4,BASE_NO 2,IPO_FRAME #BASE,POINT2[] " "}
DECL LDAT LCPDAT31={VEL 2,ACC 100.000,APO_DIST 500.000,APO_FAC 50.0000,AXIS_VEL 100.000,AXIS_ACC 100.000,ORI_TYP #VAR,CIRC_TYP #BASE,JERK_FAC 50.0000,GEAR_JERK 100.000,EXAX_IGN 0}

DECL E6POS XP32={X -233.5,Y -33.5,Z 80,A 0,B -45,C 180,S 6,T 16,E1 0.0,E2 0.0,E3 0.0,E4 0.0,E5 0.0,E6 0.0}
DECL FDAT FP32={TOOL_NO 4,BASE_NO 2,IPO_FRAME #BASE,POINT2[] " "}
DECL LDAT LCPDAT32={VEL 2,ACC 100.000,APO_DIST 500.000,APO_FAC 50.0000,AXIS_VEL 100.000,AXIS_ACC 100.000,ORI_TYP #VAR,CIRC_TYP #BASE,JERK_FAC 50.0000,GEAR_JERK 100.000,EXAX_IGN 0}

DECL E6POS XP33={X -233.5,Y 6.5,Z 80,A 0,B -45,C 180,S 6,T 16,E1 0.0,E2 0.0,E3 0.0,E4 0.0,E5 0.0,E6 0.0}
DECL FDAT FP33={TOOL_NO 4,BASE_NO 2,IPO_FRAME #BASE,POINT2[] " "}
DECL LDAT LCPDAT33={VEL 2,ACC 100.000,APO_DIST 500.000,APO_FAC 50.0000,AXIS_VEL 100.000,AXIS_ACC 100.000,ORI_TYP #VAR,CIRC_TYP #BASE,JERK_FAC 50.0000,GEAR_JERK 100.000,EXAX_IGN 0}

DECL E6POS XP34={X -233.5,Y 46.5,Z 80,A 0,B -45,C 180,S 6,T 16,E1 0.0,E2 0.0,E3 0.0,E4 0.0,E5 0.0,E6 0.0}
DECL FDAT FP34={TOOL_NO 4,BASE_NO 2,IPO_FRAME #BASE,POINT2[] " "}
DECL LDAT LCPDAT34={VEL 2,ACC 100.000,APO_DIST 500.000,APO_FAC 50.0000,AXIS_VEL 100.000,AXIS_ACC 100.000,ORI_TYP #VAR,CIRC_TYP #BASE,JERK_FAC 50.0000,GEAR_JERK 100.000,EXAX_IGN 0}

DECL E6POS XP35={X -233.5,Y 86.5,Z 80,A 0,B -45,C 180,S 6,T 16,E1 0.0,E2 0.0,E3 0.0,E4 0.0,E5 0.0,E6 0.0}
DECL FDAT FP35={TOOL_NO 4,BASE_NO 2,IPO_FRAME #BASE,POINT2[] " "}
DECL LDAT LCPDAT35={VEL 2,ACC 100.000,APO_DIST 500.000,APO_FAC 50.0000,AXIS_VEL 100.000,AXIS_ACC 100.000,ORI_TYP #VAR,CIRC_TYP #BASE,JERK_FAC 50.0000,GEAR_JERK 100.000,EXAX_IGN 0}

DECL E6POS XP36={X -233.5,Y 126.5,Z 80,A 0,B -45,C 180,S 6,T 16,E1 0.0,E2 0.0,E3 0.0,E4 0.0,E5 0.0,E6 0.0}
DECL FDAT FP36={TOOL_NO 4,BASE_NO 2,IPO_FRAME #BASE,POINT2[] " "}
DECL LDAT LCPDAT36={VEL 2,ACC 100.000,APO_DIST 500.000,APO_FAC 50.0000,AXIS_VEL 100.000,AXIS_ACC 100.000,ORI_TYP #VAR,CIRC_TYP #BASE,JERK_FAC 50.0000,GEAR_JERK 100.000,EXAX_IGN 0}

DECL E6POS XP37={X -233.5,Y 166.5,Z 80,A 0,B -45,C 180,S 6,T 16,E1 0.0,E2 0.0,E3 0.0,E4 0.0,E5 0.0,E6 0.0}
DECL FDAT FP37={TOOL_NO 4,BASE_NO 2,IPO_FRAME #BASE,POINT2[] " "}
DECL LDAT LCPDAT37={VEL 2,ACC 100.000,APO_DIST 500.000,APO_FAC 50.0000,AXIS_VEL 100.000,AXIS_ACC 100.000,ORI_TYP #VAR,CIRC_TYP #BASE,JERK_FAC 50.0000,GEAR_JERK 100.000,EXAX_IGN 0}

DECL E6POS XP38={X -233.5,Y 206.5,Z 80,A 0,B -45,C 180,S 6,T 16,E1 0.0,E2 0.0,E3 0.0,E4 0.0,E5 0.0,E6 0.0}
DECL FDAT FP38={TOOL_NO 4,BASE_NO 2,IPO_FRAME #BASE,POINT2[] " "}
DECL LDAT LCPDAT38={VEL 2,ACC 100.000,APO_DIST 500.000,APO_FAC 50.0000,AXIS_VEL 100.000,AXIS_ACC 100.000,ORI_TYP #VAR,CIRC_TYP #BASE,JERK_FAC 50.0000,GEAR_JERK 100.000,EXAX_IGN 0}

DECL E6POS XP39={X -233.5,Y 206.5,Z 120,A 0,B -45,C 180,S 6,T 16,E1 0.0,E2 0.0,E3 0.0,E4 0.0,E5 0.0,E6 0.0}
DECL FDAT FP39={TOOL_NO 4,BASE_NO 2,IPO_FRAME #BASE,POINT2[] " "}
DECL LDAT LCPDAT39={VEL 2,ACC 100.000,APO_DIST 500.000,APO_FAC 50.0000,AXIS_VEL 100.000,AXIS_ACC 100.000,ORI_TYP #VAR,CIRC_TYP #BASE,JERK_FAC 50.0000,GEAR_JERK 100.000,EXAX_IGN 0}

DECL E6POS XP40={X -233.5,Y 166.5,Z 120,A 0,B -45,C 180,S 6,T 16,E1 0.0,E2 0.0,E3 0.0,E4 0.0,E5 0.0,E6 0.0}
DECL FDAT FP40={TOOL_NO 4,BASE_NO 2,IPO_FRAME #BASE,POINT2[] " "}
DECL LDAT LCPDAT40={VEL 2,ACC 100.000,APO_DIST 500.000,APO_FAC 50.0000,AXIS_VEL 100.000,AXIS_ACC 100.000,ORI_TYP #VAR,CIRC_TYP #BASE,JERK_FAC 50.0000,GEAR_JERK 100.000,EXAX_IGN 0}

DECL E6POS XP41={X -233.5,Y 126.5,Z 120,A 0,B -45,C 180,S 6,T 16,E1 0.0,E2 0.0,E3 0.0,E4 0.0,E5 0.0,E6 0.0}
DECL FDAT FP41={TOOL_NO 4,BASE_NO 2,IPO_FRAME #BASE,POINT2[] " "}
DECL LDAT LCPDAT41={VEL 2,ACC 100.000,APO_DIST 500.000,APO_FAC 50.0000,AXIS_VEL 100.000,AXIS_ACC 100.000,ORI_TYP #VAR,CIRC_TYP #BASE,JERK_FAC 50.0000,GEAR_JERK 100.000,EXAX_IGN 0}

DECL E6POS XP42={X -233.5,Y 86.5,Z 120,A 0,B -45,C 180,S 6,T 16,E1 0.0,E2 0.0,E3 0.0,E4 0.0,E5 0.0,E6 0.0}
DECL FDAT FP42={TOOL_NO 4,BASE_NO 2,IPO_FRAME #BASE,POINT2[] " "}
DECL LDAT LCPDAT42={VEL 2,ACC 100.000,APO_DIST 500.000,APO_FAC 50.0000,AXIS_VEL 100.000,AXIS_ACC 100.000,ORI_TYP #VAR,CIRC_TYP #BASE,JERK_FAC 50.0000,GEAR_JERK 100.000,EXAX_IGN 0}

DECL E6POS XP43={X -233.5,Y 46.5,Z 120,A 0,B -45,C 180,S 6,T 16,E1 0.0,E2 0.0,E3 0.0,E4 0.0,E5 0.0,E6 0.0}
DECL FDAT FP43={TOOL_NO 4,BASE_NO 2,IPO_FRAME #BASE,POINT2[] " "}
DECL LDAT LCPDAT43={VEL 2,ACC 100.000,APO_DIST 500.000,APO_FAC 50.0000,AXIS_VEL 100.000,AXIS_ACC 100.000,ORI_TYP #VAR,CIRC_TYP #BASE,JERK_FAC 50.0000,GEAR_JERK 100.000,EXAX_IGN 0}

DECL E6POS XP44={X -233.5,Y 6.5,Z 120,A 0,B -45,C 180,S 6,T 16,E1 0.0,E2 0.0,E3 0.0,E4 0.0,E5 0.0,E6 0.0}
DECL FDAT FP44={TOOL_NO 4,BASE_NO 2,IPO_FRAME #BASE,POINT2[] " "}
DECL LDAT LCPDAT44={VEL 2,ACC 100.000,APO_DIST 500.000,APO_FAC 50.0000,AXIS_VEL 100.000,AXIS_ACC 100.000,ORI_TYP #VAR,CIRC_TYP #BASE,JERK_FAC 50.0000,GEAR_JERK 100.000,EXAX_IGN 0}

DECL E6POS XP45={X -233.5,Y -33.5,Z 120,A 0,B -45,C 180,S 6,T 16,E1 0.0,E2 0.0,E3 0.0,E4 0.0,E5 0.0,E6 0.0}
DECL FDAT FP45={TOOL_NO 4,BASE_NO 2,IPO_FRAME #BASE,POINT2[] " "}
DECL LDAT LCPDAT45={VEL 2,ACC 100.000,APO_DIST 500.000,APO_FAC 50.0000,AXIS_VEL 100.000,AXIS_ACC 100.000,ORI_TYP #VAR,CIRC_TYP #BASE,JERK_FAC 50.0000,GEAR_JERK 100.000,EXAX_IGN 0}

DECL E6POS XP46={X -233.5,Y -73.5,Z 120,A 0,B -45,C 180,S 6,T 16,E1 0.0,E2 0.0,E3 0.0,E4 0.0,E5 0.0,E6 0.0}
DECL FDAT FP46={TOOL_NO 4,BASE_NO 2,IPO_FRAME #BASE,POINT2[] " "}
DECL LDAT LCPDAT46={VEL 2,ACC 100.000,APO_DIST 500.000,APO_FAC 50.0000,AXIS_VEL 100.000,AXIS_ACC 100.000,ORI_TYP #VAR,CIRC_TYP #BASE,JERK_FAC 50.0000,GEAR_JERK 100.000,EXAX_IGN 0}

DECL E6POS XP47={X -233.5,Y -113.5,Z 120,A 0,B -45,C 180,S 6,T 16,E1 0.0,E2 0.0,E3 0.0,E4 0.0,E5 0.0,E6 0.0}
DECL FDAT FP47={TOOL_NO 4,BASE_NO 2,IPO_FRAME #BASE,POINT2[] " "}
DECL LDAT LCPDAT47={VEL 2,ACC 100.000,APO_DIST 500.000,APO_FAC 50.0000,AXIS_VEL 100.000,AXIS_ACC 100.000,ORI_TYP #VAR,CIRC_TYP #BASE,JERK_FAC 50.0000,GEAR_JERK 100.000,EXAX_IGN 0}

DECL E6POS XP48={X -233.5,Y -153.5,Z 120,A 0,B -45,C 180,S 6,T 16,E1 0.0,E2 0.0,E3 0.0,E4 0.0,E5 0.0,E6 0.0}
DECL FDAT FP48={TOOL_NO 4,BASE_NO 2,IPO_FRAME #BASE,POINT2[] " "}
DECL LDAT LCPDAT48={VEL 2,ACC 100.000,APO_DIST 500.000,APO_FAC 50.0000,AXIS_VEL 100.000,AXIS_ACC 100.000,ORI_TYP #VAR,CIRC_TYP #BASE,JERK_FAC 50.0000,GEAR_JERK 100.000,EXAX_IGN 0}

DECL E6POS XP49={X -233.5,Y -193.5,Z 120,A 0,B -45,C 180,S 6,T 16,E1 0.0,E2 0.0,E3 0.0,E4 0.0,E5 0.0,E6 0.0}
DECL FDAT FP49={TOOL_NO 4,BASE_NO 2,IPO_FRAME #BASE,POINT2[] " "}
DECL LDAT LCPDAT49={VEL 2,ACC 100.000,APO_DIST 500.000,APO_FAC 50.0000,AXIS_VEL 100.000,AXIS_ACC 100.000,ORI_TYP #VAR,CIRC_TYP #BASE,JERK_FAC 50.0000,GEAR_JERK 100.000,EXAX_IGN 0}

DECL E6POS XP50={X -233.5,Y -233.5,Z 120,A 0,B -45,C 180,S 6,T 16,E1 0.0,E2 0.0,E3 0.0,E4 0.0,E5 0.0,E6 0.0}
DECL FDAT FP50={TOOL_NO 4,BASE_NO 2,IPO_FRAME #BASE,POINT2[] " "}
DECL LDAT LCPDAT50={VEL 2,ACC 100.000,APO_DIST 500.000,APO_FAC 50.0000,AXIS_VEL 100.000,AXIS_ACC 100.000,ORI_TYP #VAR,CIRC_TYP #BASE,JERK_FAC 50.0000,GEAR_JERK 100.000,EXAX_IGN 0}

DECL E6POS XP51={X -233.5,Y -233.5,Z 160,A 0,B -45,C 180,S 6,T 16,E1 0.0,E2 0.0,E3 0.0,E4 0.0,E5 0.0,E6 0.0}
DECL FDAT FP51={TOOL_NO 4,BASE_NO 2,IPO_FRAME #BASE,POINT2[] " "}
DECL LDAT LCPDAT51={VEL 2,ACC 100.000,APO_DIST 500.000,APO_FAC 50.0000,AXIS_VEL 100.000,AXIS_ACC 100.000,ORI_TYP #VAR,CIRC_TYP #BASE,JERK_FAC 50.0000,GEAR_JERK 100.000,EXAX_IGN 0}

DECL E6POS XP52={X -233.5,Y -193.5,Z 160,A 0,B -45,C 180,S 6,T 16,E1 0.0,E2 0.0,E3 0.0,E4 0.0,E5 0.0,E6 0.0}
DECL FDAT FP52={TOOL_NO 4,BASE_NO 2,IPO_FRAME #BASE,POINT2[] " "}
DECL LDAT LCPDAT52={VEL 2,ACC 100.000,APO_DIST 500.000,APO_FAC 50.0000,AXIS_VEL 100.000,AXIS_ACC 100.000,ORI_TYP #VAR,CIRC_TYP #BASE,JERK_FAC 50.0000,GEAR_JERK 100.000,EXAX_IGN 0}

DECL E6POS XP53={X -233.5,Y -153.5,Z 160,A 0,B -45,C 180,S 6,T 16,E1 0.0,E2 0.0,E3 0.0,E4 0.0,E5 0.0,E6 0.0}
DECL FDAT FP53={TOOL_NO 4,BASE_NO 2,IPO_FRAME #BASE,POINT2[] " "}
DECL LDAT LCPDAT53={VEL 2,ACC 100.000,APO_DIST 500.000,APO_FAC 50.0000,AXIS_VEL 100.000,AXIS_ACC 100.000,ORI_TYP #VAR,CIRC_TYP #BASE,JERK_FAC 50.0000,GEAR_JERK 100.000,EXAX_IGN 0}

DECL E6POS XP54={X -233.5,Y -113.5,Z 160,A 0,B -45,C 180,S 6,T 16,E1 0.0,E2 0.0,E3 0.0,E4 0.0,E5 0.0,E6 0.0}
DECL FDAT FP54={TOOL_NO 4,BASE_NO 2,IPO_FRAME #BASE,POINT2[] " "}
DECL LDAT LCPDAT54={VEL 2,ACC 100.000,APO_DIST 500.000,APO_FAC 50.0000,AXIS_VEL 100.000,AXIS_ACC 100.000,ORI_TYP #VAR,CIRC_TYP #BASE,JERK_FAC 50.0000,GEAR_JERK 100.000,EXAX_IGN 0}

DECL E6POS XP55={X -233.5,Y -73.5,Z 160,A 0,B -45,C 180,S 6,T 16,E1 0.0,E2 0.0,E3 0.0,E4 0.0,E5 0.0,E6 0.0}
DECL FDAT FP55={TOOL_NO 4,BASE_NO 2,IPO_FRAME #BASE,POINT2[] " "}
DECL LDAT LCPDAT55={VEL 2,ACC 100.000,APO_DIST 500.000,APO_FAC 50.0000,AXIS_VEL 100.000,AXIS_ACC 100.000,ORI_TYP #VAR,CIRC_TYP #BASE,JERK_FAC 50.0000,GEAR_JERK 100.000,EXAX_IGN 0}

DECL E6POS XP56={X -233.5,Y -33.5,Z 160,A 0,B -45,C 180,S 6,T 16,E1 0.0,E2 0.0,E3 0.0,E4 0.0,E5 0.0,E6 0.0}
DECL FDAT FP56={TOOL_NO 4,BASE_NO 2,IPO_FRAME #BASE,POINT2[] " "}
DECL LDAT LCPDAT56={VEL 2,ACC 100.000,APO_DIST 500.000,APO_FAC 50.0000,AXIS_VEL 100.000,AXIS_ACC 100.000,ORI_TYP #VAR,CIRC_TYP #BASE,JERK_FAC 50.0000,GEAR_JERK 100.000,EXAX_IGN 0}

DECL E6POS XP57={X -233.5,Y 6.5,Z 160,A 0,B -45,C 180,S 6,T 16,E1 0.0,E2 0.0,E3 0.0,E4 0.0,E5 0.0,E6 0.0}
DECL FDAT FP57={TOOL_NO 4,BASE_NO 2,IPO_FRAME #BASE,POINT2[] " "}
DECL LDAT LCPDAT57={VEL 2,ACC 100.000,APO_DIST 500.000,APO_FAC 50.0000,AXIS_VEL 100.000,AXIS_ACC 100.000,ORI_TYP #VAR,CIRC_TYP #BASE,JERK_FAC 50.0000,GEAR_JERK 100.000,EXAX_IGN 0}

DECL E6POS XP58={X -233.5,Y 46.5,Z 160,A 0,B -45,C 180,S 6,T 16,E1 0.0,E2 0.0,E3 0.0,E4 0.0,E5 0.0,E6 0.0}
DECL FDAT FP58={TOOL_NO 4,BASE_NO 2,IPO_FRAME #BASE,POINT2[] " "}
DECL LDAT LCPDAT58={VEL 2,ACC 100.000,APO_DIST 500.000,APO_FAC 50.0000,AXIS_VEL 100.000,AXIS_ACC 100.000,ORI_TYP #VAR,CIRC_TYP #BASE,JERK_FAC 50.0000,GEAR_JERK 100.000,EXAX_IGN 0}

DECL E6POS XP59={X -233.5,Y 86.5,Z 160,A 0,B -45,C 180,S 6,T 16,E1 0.0,E2 0.0,E3 0.0,E4 0.0,E5 0.0,E6 0.0}
DECL FDAT FP59={TOOL_NO 4,BASE_NO 2,IPO_FRAME #BASE,POINT2[] " "}
DECL LDAT LCPDAT59={VEL 2,ACC 100.000,APO_DIST 500.000,APO_FAC 50.0000,AXIS_VEL 100.000,AXIS_ACC 100.000,ORI_TYP #VAR,CIRC_TYP #BASE,JERK_FAC 50.0000,GEAR_JERK 100.000,EXAX_IGN 0}

DECL E6POS XP60={X -233.5,Y 126.5,Z 160,A 0,B -45,C 180,S 6,T 16,E1 0.0,E2 0.0,E3 0.0,E4 0.0,E5 0.0,E6 0.0}
DECL FDAT FP60={TOOL_NO 4,BASE_NO 2,IPO_FRAME #BASE,POINT2[] " "}
DECL LDAT LCPDAT60={VEL 2,ACC 100.000,APO_DIST 500.000,APO_FAC 50.0000,AXIS_VEL 100.000,AXIS_ACC 100.000,ORI_TYP #VAR,CIRC_TYP #BASE,JERK_FAC 50.0000,GEAR_JERK 100.000,EXAX_IGN 0}

DECL E6POS XP61={X -233.5,Y 166.5,Z 160,A 0,B -45,C 180,S 6,T 16,E1 0.0,E2 0.0,E3 0.0,E4 0.0,E5 0.0,E6 0.0}
DECL FDAT FP61={TOOL_NO 4,BASE_NO 2,IPO_FRAME #BASE,POINT2[] " "}
DECL LDAT LCPDAT61={VEL 2,ACC 100.000,APO_DIST 500.000,APO_FAC 50.0000,AXIS_VEL 100.000,AXIS_ACC 100.000,ORI_TYP #VAR,CIRC_TYP #BASE,JERK_FAC 50.0000,GEAR_JERK 100.000,EXAX_IGN 0}

DECL E6POS XP62={X -233.5,Y 206.5,Z 160,A 0,B -45,C 180,S 6,T 16,E1 0.0,E2 0.0,E3 0.0,E4 0.0,E5 0.0,E6 0.0}
DECL FDAT FP62={TOOL_NO 4,BASE_NO 2,IPO_FRAME #BASE,POINT2[] " "}
DECL LDAT LCPDAT62={VEL 2,ACC 100.000,APO_DIST 500.000,APO_FAC 50.0000,AXIS_VEL 100.000,AXIS_ACC 100.000,ORI_TYP #VAR,CIRC_TYP #BASE,JERK_FAC 50.0000,GEAR_JERK 100.000,EXAX_IGN 0}

DECL E6POS XP63={X -233.5,Y 206.5,Z 200,A 0,B -45,C 180,S 6,T 16,E1 0.0,E2 0.0,E3 0.0,E4 0.0,E5 0.0,E6 0.0}
DECL FDAT FP63={TOOL_NO 4,BASE_NO 2,IPO_FRAME #BASE,POINT2[] " "}
DECL LDAT LCPDAT63={VEL 2,ACC 100.000,APO_DIST 500.000,APO_FAC 50.0000,AXIS_VEL 100.000,AXIS_ACC 100.000,ORI_TYP #VAR,CIRC_TYP #BASE,JERK_FAC 50.0000,GEAR_JERK 100.000,EXAX_IGN 0}

DECL E6POS XP64={X -233.5,Y 166.5,Z 200,A 0,B -45,C 180,S 6,T 16,E1 0.0,E2 0.0,E3 0.0,E4 0.0,E5 0.0,E6 0.0}
DECL FDAT FP64={TOOL_NO 4,BASE_NO 2,IPO_FRAME #BASE,POINT2[] " "}
DECL LDAT LCPDAT64={VEL 2,ACC 100.000,APO_DIST 500.000,APO_FAC 50.0000,AXIS_VEL 100.000,AXIS_ACC 100.000,ORI_TYP #VAR,CIRC_TYP #BASE,JERK_FAC 50.0000,GEAR_JERK 100.000,EXAX_IGN 0}

DECL E6POS XP65={X -233.5,Y 126.5,Z 200,A 0,B -45,C 180,S 6,T 16,E1 0.0,E2 0.0,E3 0.0,E4 0.0,E5 0.0,E6 0.0}
DECL FDAT FP65={TOOL_NO 4,BASE_NO 2,IPO_FRAME #BASE,POINT2[] " "}
DECL LDAT LCPDAT65={VEL 2,ACC 100.000,APO_DIST 500.000,APO_FAC 50.0000,AXIS_VEL 100.000,AXIS_ACC 100.000,ORI_TYP #VAR,CIRC_TYP #BASE,JERK_FAC 50.0000,GEAR_JERK 100.000,EXAX_IGN 0}

DECL E6POS XP66={X -233.5,Y 86.5,Z 200,A 0,B -45,C 180,S 6,T 16,E1 0.0,E2 0.0,E3 0.0,E4 0.0,E5 0.0,E6 0.0}
DECL FDAT FP66={TOOL_NO 4,BASE_NO 2,IPO_FRAME #BASE,POINT2[] " "}
DECL LDAT LCPDAT66={VEL 2,ACC 100.000,APO_DIST 500.000,APO_FAC 50.0000,AXIS_VEL 100.000,AXIS_ACC 100.000,ORI_TYP #VAR,CIRC_TYP #BASE,JERK_FAC 50.0000,GEAR_JERK 100.000,EXAX_IGN 0}

DECL E6POS XP67={X -233.5,Y 46.5,Z 200,A 0,B -45,C 180,S 6,T 16,E1 0.0,E2 0.0,E3 0.0,E4 0.0,E5 0.0,E6 0.0}
DECL FDAT FP67={TOOL_NO 4,BASE_NO 2,IPO_FRAME #BASE,POINT2[] " "}
DECL LDAT LCPDAT67={VEL 2,ACC 100.000,APO_DIST 500.000,APO_FAC 50.0000,AXIS_VEL 100.000,AXIS_ACC 100.000,ORI_TYP #VAR,CIRC_TYP #BASE,JERK_FAC 50.0000,GEAR_JERK 100.000,EXAX_IGN 0}

DECL E6POS XP68={X -233.5,Y 6.5,Z 200,A 0,B -45,C 180,S 6,T 16,E1 0.0,E2 0.0,E3 0.0,E4 0.0,E5 0.0,E6 0.0}
DECL FDAT FP68={TOOL_NO 4,BASE_NO 2,IPO_FRAME #BASE,POINT2[] " "}
DECL LDAT LCPDAT68={VEL 2,ACC 100.000,APO_DIST 500.000,APO_FAC 50.0000,AXIS_VEL 100.000,AXIS_ACC 100.000,ORI_TYP #VAR,CIRC_TYP #BASE,JERK_FAC 50.0000,GEAR_JERK 100.000,EXAX_IGN 0}

DECL E6POS XP69={X -233.5,Y -33.5,Z 200,A 0,B -45,C 180,S 6,T 16,E1 0.0,E2 0.0,E3 0.0,E4 0.0,E5 0.0,E6 0.0}
DECL FDAT FP69={TOOL_NO 4,BASE_NO 2,IPO_FRAME #BASE,POINT2[] " "}
DECL LDAT LCPDAT69={VEL 2,ACC 100.000,APO_DIST 500.000,APO_FAC 50.0000,AXIS_VEL 100.000,AXIS_ACC 100.000,ORI_TYP #VAR,CIRC_TYP #BASE,JERK_FAC 50.0000,GEAR_JERK 100.000,EXAX_IGN 0}

DECL E6POS XP70={X -233.5,Y -73.5,Z 200,A 0,B -45,C 180,S 6,T 16,E1 0.0,E2 0.0,E3 0.0,E4 0.0,E5 0.0,E6 0.0}
DECL FDAT FP70={TOOL_NO 4,BASE_NO 2,IPO_FRAME #BASE,POINT2[] " "}
DECL LDAT LCPDAT70={VEL 2,ACC 100.000,APO_DIST 500.000,APO_FAC 50.0000,AXIS_VEL 100.000,AXIS_ACC 100.000,ORI_TYP #VAR,CIRC_TYP #BASE,JERK_FAC 50.0000,GEAR_JERK 100.000,EXAX_IGN 0}

DECL E6POS XP71={X -233.5,Y -113.5,Z 200,A 0,B -45,C 180,S 6,T 16,E1 0.0,E2 0.0,E3 0.0,E4 0.0,E5 0.0,E6 0.0}
DECL FDAT FP71={TOOL_NO 4,BASE_NO 2,IPO_FRAME #BASE,POINT2[] " "}
DECL LDAT LCPDAT71={VEL 2,ACC 100.000,APO_DIST 500.000,APO_FAC 50.0000,AXIS_VEL 100.000,AXIS_ACC 100.000,ORI_TYP #VAR,CIRC_TYP #BASE,JERK_FAC 50.0000,GEAR_JERK 100.000,EXAX_IGN 0}

DECL E6POS XP72={X -233.5,Y -153.5,Z 200,A 0,B -45,C 180,S 6,T 16,E1 0.0,E2 0.0,E3 0.0,E4 0.0,E5 0.0,E6 0.0}
DECL FDAT FP72={TOOL_NO 4,BASE_NO 2,IPO_FRAME #BASE,POINT2[] " "}
DECL LDAT LCPDAT72={VEL 2,ACC 100.000,APO_DIST 500.000,APO_FAC 50.0000,AXIS_VEL 100.000,AXIS_ACC 100.000,ORI_TYP #VAR,CIRC_TYP #BASE,JERK_FAC 50.0000,GEAR_JERK 100.000,EXAX_IGN 0}

